  MoveL 3156 to (42.98, 34.27, 135) mm, rotated rx 180 ry 0 rz 180 deg; joints [33.282, 51.26, 5.095, -141.744, 62.408, -200.063]
  Call Extruder(29635.551)
  MoveL 3157 to (34.27, 42.98, 135) mm, rotated rx 180 ry 0 rz 180 deg; joints [34.874, 50.898, 5.796, -140.175, 63.224, -200.59]
  Call Extruder(29646.481)
  MoveL 3158 to (23.85, 49.52, 135) mm, rotated rx -180 ry 0 rz -180 deg; joints [36.387, 50.182, 7.18, -138.811, 64.267, -200.804]
  Call Extruder(29657.411)
  MoveL 3159 to (12.23, 53.59, 135) mm, rotated rx 180 ry 0 rz -180 deg; joints [37.766, 49.152, 9.175, -137.688, 65.475, -200.699]
  Call Extruder(29668.342)
  MoveL 3160 to (0, 54.97, 135) mm, rotated rx 180 ry 0 rz -180 deg; joints [38.954, 47.859, 11.678, -136.834, 66.781, -200.294]
  Call Extruder(29679.272)
  MoveL 3161 to (-12.23, 53.59, 135) mm, rotated rx 180 ry 0 rz -180 deg; joints [39.895, 46.371, 14.565, -136.276, 68.117, -199.62]
  Call Extruder(29690.202)
  MoveL 3162 to (-23.85, 49.53, 135) mm, rotated rx 180 ry 0 rz 180 deg; joints [40.528, 44.756, 17.699, -136.043, 69.421, -198.723]
  Call Extruder(29701.132)
  MoveL 3163 to (-34.27, 42.98, 135) mm, rotated rx 180 ry 0 rz 180 deg; joints [40.799, 43.092, 20.933, -136.165, 70.637, -197.658]
  Call Extruder(29712.062)
  MoveL 3164 to (-42.98, 34.27, 135) mm, rotated rx -180 ry 0 rz -180 deg; joints [40.659, 41.457, 24.115, -136.671, 71.717, -196.485]
  Call Extruder(29722.993)
  MoveL 3165 to (-49.53, 23.85, 135) mm, rotated rx 180 ry 0 rz 180 deg; joints [40.072, 39.93, 27.092, -137.58, 72.618, -195.268]
  Call Extruder(29733.923)
  MoveL 3166 to (-53.59, 12.23, 135) mm, rotated rx 180 ry 0 rz -180 deg; joints [39.031, 38.588, 29.712, -138.895, 73.308, -194.069]
  Call Extruder(29744.853)
  MoveL 3167 to (-54.97, 0, 135) mm, rotated rx 180 ry 0 rz -180 deg; joints [37.56, 37.502, 31.833, -140.584, 73.755, -192.948]
  Call Extruder(29750.379)
  MoveL 3168 to (-54.27, -6.18, 135) mm, rotated rx 180 ry 0 rz -180 deg; joints [36.644, 37.108, 32.604, -141.583, 73.846, -192.442]
  Set speed (130.0 mm/s)
  MoveL 3169 to (-49.9, -9.51, 135) mm, rotated rx -180 ry 0 rz 180 deg; joints [35.741, 37.302, 32.224, -142.469, 73.507, -192.303]
  MoveL 3170 to (2.97, -12.99, 135) mm, rotated rx 180 ry 0 rz -180 deg; joints [30.614, 42.764, 21.571, -146.715, 68.115, -193.75]
  Call Extruder(29755.042)
  Set speed (80.0 mm/s)
  MoveL 3171 to (5.78, -12.01, 135) mm, rotated rx -180 ry 0 rz -180 deg; joints [30.526, 43.158, 20.805, -146.725, 67.783, -193.936]
  Call Extruder(29759.706)
  MoveL 3172 to (8.31, -10.42, 135) mm, rotated rx -180 ry 0 rz -180 deg; joints [30.538, 43.562, 20.019, -146.625, 67.467, -194.168]
  Call Extruder(29764.370)
  MoveL 3173 to (10.42, -8.31, 135) mm, rotated rx 180 ry 0 rz 180 deg; joints [30.649, 43.956, 19.253, -146.423, 67.184, -194.435]
  Call Extruder(29769.034)
  MoveL 3174 to (12.01, -5.78, 135) mm, rotated rx 180 ry 0 rz -180 deg; joints [30.85, 44.321, 18.544, -146.131, 66.949, -194.725]
  Call Extruder(29773.697)
  MoveL 3175 to (12.99, -2.97, 135) mm, rotated rx 180 ry 0 rz -180 deg; joints [31.131, 44.637, 17.929, -145.765, 66.773, -195.022]
  Call Extruder(29778.361)
  MoveL 3176 to (13.33, 0, 135) mm, rotated rx 180 ry 0 rz -180 deg; joints [31.476, 44.891, 17.438, -145.344, 66.667, -195.312]
  Call Extruder(29783.025)
  MoveL 3177 to (12.99, 2.97, 135) mm, rotated rx 180 ry 0 rz -180 deg; joints [31.869, 45.068, 17.094, -144.89, 66.635, -195.58]
  Call Extruder(29787.689)
  MoveL 3178 to (12.01, 5.78, 135) mm, rotated rx 180 ry 0 rz -180 deg; joints [32.292, 45.16, 16.915, -144.425, 66.679, -195.81]
  Call Extruder(29792.352)
  MoveL 3179 to (10.42, 8.31, 135) mm, rotated rx 180 ry 0 rz 180 deg; joints [32.725, 45.162, 16.91, -143.971, 66.795, -195.991]
  Call Extruder(29797.017)
  MoveL 3180 to (8.31, 10.42, 135) mm, rotated rx -180 ry 0 rz -180 deg; joints [33.149, 45.075, 17.079, -143.549, 66.978, -196.112]
  Call Extruder(29801.680)
  MoveL 3181 to (5.78, 12.01, 135) mm, rotated rx 180 ry 0 rz -180 deg; joints [33.544, 44.903, 17.413, -143.177, 67.219, -196.167]
  Call Extruder(29806.344)
  MoveL 3182 to (2.97, 13, 135) mm, rotated rx 180 ry 0 rz -180 deg; joints [33.893, 44.654, 17.897, -142.874, 67.503, -196.154]
  Call Extruder(29811.008)
  MoveL 3183 to (0, 13.33, 135) mm, rotated rx 180 ry 0 rz 180 deg; joints [34.177, 44.341, 18.505, -142.652, 67.817, -196.073]
  Call Extruder(29815.672)
  MoveL 3184 to (-2.97, 12.99, 135) mm, rotated rx -180 ry 0 rz 180 deg; joints [34.384, 43.979, 19.209, -142.522, 68.145, -195.93]
  Call Extruder(29820.335)
  MoveL 3185 to (-5.78, 12.01, 135) mm, rotated rx 180 ry 0 rz 180 deg; joints [34.5, 43.586, 19.973, -142.491, 68.471, -195.731]
  Call Extruder(29824.999)
  MoveL 3186 to (-8.31, 10.42, 135) mm, rotated rx 180 ry 0 rz 180 deg; joints [34.518, 43.182, 20.759, -142.563, 68.779, -195.489]
  Call Extruder(29829.663)
  MoveL 3187 to (-10.42, 8.31, 135) mm, rotated rx 180 ry 0 rz -180 deg; joints [34.436, 42.787, 21.527, -142.735, 69.054, -195.215]
  Call Extruder(29834.327)
  MoveL 3188 to (-12.01, 5.78, 135) mm, rotated rx 180 ry 0 rz 180 deg; joints [34.254, 42.42, 22.24, -143.003, 69.283, -194.925]
  Call Extruder(29838.990)
  MoveL 3189 to (-12.99, 2.97, 135) mm, rotated rx 180 ry 0 rz 180 deg; joints [33.981, 42.101, 22.861, -143.353, 69.455, -194.632]
  Call Extruder(29843.654)
  MoveL 3190 to (-13.33, 0, 135) mm, rotated rx 180 ry 0 rz 180 deg; joints [33.63, 41.846, 23.359, -143.77, 69.562, -194.351]
  Call Extruder(29848.318)
  MoveL 3191 to (-13, -2.97, 135) mm, rotated rx 180 ry 0 rz -180 deg; joints [33.218, 41.667, 23.707, -144.233, 69.598, -194.096]
  Call Extruder(29852.982)
  MoveL 3192 to (-12.01, -5.78, 135) mm, rotated rx 180 ry 0 rz 180 deg; joints [32.767, 41.573, 23.889, -144.719, 69.561, -193.879]
  Call Extruder(29857.645)
  MoveL 3193 to (-10.42, -8.31, 135) mm, rotated rx 180 ry 0 rz 180 deg; joints [32.302, 41.571, 23.894, -145.201, 69.452, -193.708]
  Call Extruder(29862.310)
  MoveL 3194 to (-8.31, -10.42, 135) mm, rotated rx -180 ry 0 rz -180 deg; joints [31.85, 41.659, 23.723, -145.653, 69.277, -193.594]
  Call Extruder(29866.973)
  MoveL 3195 to (-5.78, -12.01, 135) mm, rotated rx 180 ry 0 rz 180 deg; joints [31.435, 41.833, 23.384, -146.05, 69.043, -193.539]
  Call Extruder(29871.637)
  MoveL 3196 to (-2.97, -12.99, 135) mm, rotated rx -180 ry 0 rz -180 deg; joints [31.079, 42.084, 22.894, -146.369, 68.762, -193.548]
  Call Extruder(29876.301)
  MoveL 3197 to (0, -13.33, 135) mm, rotated rx 180 ry 0 rz -180 deg; joints [30.801, 42.4, 22.279, -146.595, 68.447, -193.619]
  Call Extruder(29880.965)
  MoveL 3198 to (2.97, -12.99, 135) mm, rotated rx 180 ry 0 rz -180 deg; joints [30.614, 42.764, 21.571, -146.715, 68.115, -193.75]
  Set speed (130.0 mm/s)
  MoveL 3199 to (2.97, -12.99, 140) mm, rotated rx -180 ry 0 rz -180 deg; joints [30.614, 41.931, 21.714, -146.56, 67.539, -194.16]
  MoveL 3200 to (-26.25, -4.54, 140) mm, rotated rx 180 ry 0 rz 180 deg; joints [34.172, 39.236, 26.879, -143.407, 70.428, -193.968]
  Call Extruder(29883.197)
  Set speed (60.0 mm/s)
  MoveL 3201 to (-26.09, -5.96, 140) mm, rotated rx 180 ry 0 rz -180 deg; joints [33.969, 39.149, 27.045, -143.633, 70.443, -193.847]
  Call Extruder(29892.562)
  MoveL 3202 to (-24.12, -11.61, 140) mm, rotated rx 180 ry 0 rz -180 deg; joints [33.033, 38.956, 27.415, -144.635, 70.366, -193.413]
  Call Extruder(29901.927)
  MoveL 3203 to (-20.93, -16.69, 140) mm, rotated rx 180 ry 0 rz 180 deg; joints [32.066, 38.951, 27.426, -145.637, 70.148, -193.072]
  Call Extruder(29911.292)
  MoveL 3204 to (-16.69, -20.93, 140) mm, rotated rx 180 ry 0 rz 180 deg; joints [31.126, 39.133, 27.077, -146.578, 69.799, -192.838]
  Call Extruder(29920.657)
  MoveL 3205 to (-11.61, -24.11, 140) mm, rotated rx -180 ry 0 rz -180 deg; joints [30.272, 39.492, 26.388, -147.4, 69.334, -192.719]
  Call Extruder(29930.022)
  MoveL 3206 to (-5.96, -26.09, 140) mm, rotated rx 180 ry 0 rz 180 deg; joints [29.552, 40.01, 25.395, -148.055, 68.774, -192.721]
  Call Extruder(29939.387)
  MoveL 3207 to (0, -26.77, 140) mm, rotated rx 180 ry 0 rz 180 deg; joints [29.003, 40.659, 24.152, -148.507, 68.146, -192.846]
  Call Extruder(29948.752)
  MoveL 3208 to (5.96, -26.09, 140) mm, rotated rx 180 ry 0 rz 180 deg; joints [28.65, 41.404, 22.723, -148.733, 67.484, -193.09]
  Call Extruder(29958.117)
  MoveL 3209 to (11.61, -24.11, 140) mm, rotated rx 180 ry 0 rz 180 deg; joints [28.503, 42.209, 21.181, -148.728, 66.819, -193.446]
  Call Extruder(29967.482)
  MoveL 3210 to (16.69, -20.93, 140) mm, rotated rx -180 ry 0 rz -180 deg; joints [28.559, 43.032, 19.602, -148.497, 66.188, -193.898]
  Call Extruder(29976.847)
  MoveL 3211 to (20.93, -16.69, 140) mm, rotated rx 180 ry 0 rz 180 deg; joints [28.808, 43.834, 18.066, -148.06, 65.624, -194.429]
  Call Extruder(29986.212)
  MoveL 3212 to (24.12, -11.61, 140) mm, rotated rx 180 ry 0 rz -180 deg; joints [29.229, 44.574, 16.648, -147.446, 65.157, -195.014]
  Call Extruder(29995.577)
  MoveL 3213 to (26.09, -5.96, 140) mm, rotated rx 180 ry 0 rz -180 deg; joints [29.796, 45.217, 15.416, -146.693, 64.813, -195.622]
  Call Extruder(30004.942)
  MoveL 3214 to (26.77, 0, 140) mm, rotated rx 180 ry 0 rz -180 deg; joints [30.482, 45.73, 14.431, -145.841, 64.609, -196.223]
  Call Extruder(30014.307)
  MoveL 3215 to (26.09, 5.96, 140) mm, rotated rx 180 ry 0 rz -180 deg; joints [31.252, 46.09, 13.743, -144.933, 64.557, -196.781]
  Call Extruder(30023.672)
  MoveL 3216 to (24.12, 11.61, 140) mm, rotated rx 180 ry 0 rz -180 deg; joints [32.076, 46.277, 13.385, -144.015, 64.659, -197.265]
  Call Extruder(30033.037)
  MoveL 3217 to (20.93, 16.69, 140) mm, rotated rx 180 ry 0 rz -180 deg; joints [32.917, 46.282, 13.374, -143.126, 64.907, -197.646]
  Call Extruder(30042.402)
  MoveL 3218 to (16.69, 20.93, 140) mm, rotated rx 180 ry 0 rz 180 deg; joints [33.742, 46.106, 13.712, -142.305, 65.288, -197.903]
  Call Extruder(30051.767)
  MoveL 3219 to (11.61, 24.12, 140) mm, rotated rx 180 ry 0 rz 180 deg; joints [34.517, 45.756, 14.382, -141.585, 65.779, -198.022]
  Call Extruder(30061.132)
  MoveL 3220 to (5.96, 26.09, 140) mm, rotated rx 180 ry 0 rz 180 deg; joints [35.208, 45.251, 15.351, -140.995, 66.354, -197.997]
  Call Extruder(30070.497)
  MoveL 3221 to (0, 26.77, 140) mm, rotated rx 180 ry 0 rz 180 deg; joints [35.784, 44.615, 16.569, -140.557, 66.983, -197.831]
  Call Extruder(30079.862)
  MoveL 3222 to (-5.96, 26.09, 140) mm, rotated rx 180 ry 0 rz 180 deg; joints [36.214, 43.879, 17.979, -140.292, 67.633, -197.537]
  Call Extruder(30089.227)
  MoveL 3223 to (-11.61, 24.12, 140) mm, rotated rx 180 ry 0 rz -180 deg; joints [36.473, 43.08, 19.51, -140.215, 68.273, -197.132]
  Call Extruder(30098.591)
  MoveL 3224 to (-16.69, 20.93, 140) mm, rotated rx 180 ry 0 rz 180 deg; joints [36.542, 42.257, 21.088, -140.334, 68.874, -196.64]
  Call Extruder(30107.957)
  MoveL 3225 to (-20.93, 16.69, 140) mm, rotated rx 180 ry 0 rz -180 deg; joints [36.407, 41.451, 22.634, -140.652, 69.406, -196.087]
  Call Extruder(30117.322)
  MoveL 3226 to (-24.12, 11.61, 140) mm, rotated rx 180 ry 0 rz 180 deg; joints [36.065, 40.7, 24.072, -141.163, 69.847, -195.502]
  Call Extruder(30126.686)
  MoveL 3227 to (-26.09, 5.96, 140) mm, rotated rx 180 ry 0 rz 180 deg; joints [35.528, 40.045, 25.328, -141.851, 70.176, -194.916]
  Call Extruder(30136.051)
  MoveL 3228 to (-26.77, 0, 140) mm, rotated rx 180 ry 0 rz 180 deg; joints [34.817, 39.519, 26.337, -142.688, 70.378, -194.355]
  Call Extruder(30140.840)
  MoveL 3229 to (-26.42, -3.05, 140) mm, rotated rx 180 ry 0 rz -180 deg; joints [34.385, 39.328, 26.702, -143.17, 70.412, -194.095]
  Set speed (130.0 mm/s)
  MoveL 3230 to (-41.86, -6.29, 140) mm, rotated rx 180 ry 0 rz -180 deg; joints [35.393, 37.441, 30.319, -142.491, 72.029, -193.324]
  Call Extruder(30145.838)
  Set speed (60.0 mm/s)
  MoveL 3231 to (-41.5, -9.47, 140) mm, rotated rx 180 ry 0 rz -180 deg; joints [34.924, 37.244, 30.696, -143.006, 72.065, -193.061]
  Call Extruder(30160.734)
  MoveL 3232 to (-38.36, -18.47, 140) mm, rotated rx 180 ry 0 rz -180 deg; joints [33.373, 36.932, 31.296, -144.652, 71.955, -192.392]
  Call Extruder(30175.630)
  MoveL 3233 to (-33.29, -26.54, 140) mm, rotated rx 180 ry 0 rz 180 deg; joints [31.763, 36.923, 31.313, -146.31, 71.624, -191.869]
  Call Extruder(30190.525)
  MoveL 3234 to (-26.54, -33.29, 140) mm, rotated rx -180 ry 0 rz 180 deg; joints [30.206, 37.218, 30.748, -147.87, 71.081, -191.509]
  Call Extruder(30205.421)
  MoveL 3235 to (-18.47, -38.36, 140) mm, rotated rx 180 ry 0 rz 180 deg; joints [28.808, 37.799, 29.633, -149.225, 70.349, -191.325]
  Call Extruder(30220.317)
  MoveL 3236 to (-9.47, -41.5, 140) mm, rotated rx 180 ry 0 rz 180 deg; joints [27.654, 38.634, 28.033, -150.288, 69.462, -191.321]
  Call Extruder(30235.213)
  MoveL 3237 to (0, -42.57, 140) mm, rotated rx -180 ry 0 rz -180 deg; joints [26.805, 39.675, 26.038, -151, 68.462, -191.502]
  Call Extruder(30250.109)
  MoveL 3238 to (9.47, -41.5, 140) mm, rotated rx 180 ry 0 rz -180 deg; joints [26.29, 40.867, 23.753, -151.331, 67.401, -191.866]
  Call Extruder(30265.004)
  MoveL 3239 to (18.47, -38.36, 140) mm, rotated rx 180 ry 0 rz 180 deg; joints [26.114, 42.149, 21.296, -151.277, 66.333, -192.407]
  Call Extruder(30279.900)
  MoveL 3240 to (26.54, -33.29, 140) mm, rotated rx -180 ry 0 rz 180 deg; joints [26.262, 43.457, 18.787, -150.858, 65.315, -193.108]
  Call Extruder(30294.796)
  MoveL 3241 to (33.28, -26.54, 140) mm, rotated rx 180 ry 0 rz 180 deg; joints [26.703, 44.73, 16.349, -150.114, 64.404, -193.944]
  Call Extruder(30309.692)
  MoveL 3242 to (38.36, -18.47, 140) mm, rotated rx 180 ry 0 rz 180 deg; joints [27.4, 45.905, 14.097, -149.098, 63.648, -194.878]
  Call Extruder(30324.587)
  MoveL 3243 to (41.51, -9.47, 140) mm, rotated rx 180 ry 0 rz 180 deg; joints [28.309, 46.926, 12.141, -147.873, 63.091, -195.865]
  Call Extruder(30339.483)
  MoveL 3244 to (42.57, 0, 140) mm, rotated rx 180 ry 0 rz 180 deg; joints [29.382, 47.743, 10.575, -146.508, 62.765, -196.847]
  Call Extruder(30354.379)
  MoveL 3245 to (41.5, 9.47, 140) mm, rotated rx 180 ry 0 rz -180 deg; joints [30.575, 48.315, 9.478, -145.076, 62.686, -197.765]
  Call Extruder(30369.275)
  MoveL 3246 to (38.36, 18.47, 140) mm, rotated rx -180 ry 0 rz -180 deg; joints [31.839, 48.614, 8.907, -143.643, 62.858, -198.563]
  Call Extruder(30384.171)
  MoveL 3247 to (33.29, 26.54, 140) mm, rotated rx 180 ry 0 rz -180 deg; joints [33.128, 48.622, 8.89, -142.273, 63.269, -199.188]
  Call Extruder(30399.067)
  MoveL 3248 to (26.54, 33.28, 140) mm, rotated rx -180 ry 0 rz -180 deg; joints [34.394, 48.341, 9.43, -141.018, 63.891, -199.603]
  Call Extruder(30413.962)
  MoveL 3249 to (18.47, 38.36, 140) mm, rotated rx -180 ry 0 rz 180 deg; joints [35.592, 47.784, 10.496, -139.922, 64.689, -199.785]
  Call Extruder(30428.858)
  MoveL 3250 to (9.47, 41.51, 140) mm, rotated rx 180 ry 0 rz -180 deg; joints [36.675, 46.98, 12.037, -139.022, 65.614, -199.73]
  Call Extruder(30443.754)
  MoveL 3251 to (0, 42.57, 140) mm, rotated rx 180 ry 0 rz 180 deg; joints [37.594, 45.97, 13.973, -138.345, 66.618, -199.445]
  Call Extruder(30458.650)
  MoveL 3252 to (-9.47, 41.51, 140) mm, rotated rx -180 ry 0 rz -180 deg; joints [38.304, 44.802, 16.21, -137.918, 67.648, -198.953]
  Call Extruder(30473.545)
  MoveL 3253 to (-18.47, 38.36, 140) mm, rotated rx 180 ry 0 rz 180 deg; joints [38.762, 43.534, 18.641, -137.763, 68.656, -198.286]
  Call Extruder(30488.441)
  MoveL 3254 to (-26.54, 33.29, 140) mm, rotated rx 180 ry 0 rz -180 deg; joints [38.928, 42.226, 21.148, -137.901, 69.596, -197.485]
  Call Extruder(30503.337)
  MoveL 3255 to (-33.28, 26.54, 140) mm, rotated rx 180 ry 0 rz 180 deg; joints [38.772, 40.941, 23.612, -138.346, 70.427, -196.594]
  Call Extruder(30518.233)
  MoveL 3256 to (-38.36, 18.47, 140) mm, rotated rx 180 ry 0 rz 180 deg; joints [38.277, 39.742, 25.91, -139.103, 71.116, -195.66]
  Call Extruder(30533.129)
  MoveL 3257 to (-41.51, 9.47, 140) mm, rotated rx 180 ry 0 rz -180 deg; joints [37.447, 38.69, 27.925, -140.159, 71.633, -194.731]
  Call Extruder(30548.024)
  MoveL 3258 to (-42.57, 0, 140) mm, rotated rx 180 ry 0 rz -180 deg; joints [36.31, 37.842, 29.551, -141.48, 71.955, -193.851]
  Call Extruder(30555.579)
  MoveL 3259 to (-42.03, -4.8, 140) mm, rotated rx -180 ry 0 rz 180 deg; joints [35.612, 37.535, 30.139, -142.25, 72.011, -193.448]
  Set speed (130.0 mm/s)
  MoveL 3260 to (-54.1, -7.67, 140) mm, rotated rx 180 ry 0 rz -180 deg; joints [36.421, 36.076, 32.935, -141.682, 73.249, -192.831]
  Call Extruder(30559.651)
  Set speed (30.0 mm/s)
  MoveL 3261 to (-53.59, -12.23, 140) mm, rotated rx 180 ry 0 rz -180 deg; joints [35.732, 35.79, 33.484, -142.433, 73.304, -192.461]
  Call Extruder(30570.582)
  MoveL 3262 to (-49.53, -23.85, 140) mm, rotated rx 180 ry 0 rz -180 deg; joints [33.663, 35.379, 34.271, -144.613, 73.176, -191.618]
  Call Extruder(30581.512)
  MoveL 3263 to (-42.98, -34.27, 140) mm, rotated rx 180 ry 0 rz 180 deg; joints [31.506, 35.367, 34.294, -146.828, 72.762, -190.963]
  Call Extruder(30592.442)
  MoveL 3264 to (-34.27, -42.98, 140) mm, rotated rx -180 ry 0 rz 180 deg; joints [29.427, 35.755, 33.55, -148.91, 72.074, -190.514]
  Call Extruder(30603.372)
  MoveL 3265 to (-23.85, -49.53, 140) mm, rotated rx -180 ry 0 rz 180 deg; joints [27.581, 36.518, 32.089, -150.707, 71.136, -190.281]
  Call Extruder(30614.302)
  MoveL 3266 to (-12.23, -53.59, 140) mm, rotated rx -180 ry 0 rz -180 deg; joints [26.087, 37.608, 29.999, -152.097, 69.992, -190.269]
  Call Extruder(30625.233)
  MoveL 3267 to (0, -54.97, 140) mm, rotated rx 180 ry 0 rz 180 deg; joints [25.019, 38.963, 27.403, -153.004, 68.698, -190.485]
  Call Extruder(30634.985)
  MoveL 3268 to (10.91, -53.74, 140) mm, rotated rx 180 ry 0 rz 180 deg; joints [24.47, 40.34, 24.764, -153.357, 67.47, -190.882]
  Call Extruder(30636.163)
  MoveL 3269 to (12.23, -53.59, 140) mm, rotated rx -180 ry 0 rz -180 deg; joints [24.406, 40.508, 24.441, -153.396, 67.32, -190.931]
  Call Extruder(30647.093)
  MoveL 3270 to (23.85, -49.52, 140) mm, rotated rx -180 ry 0 rz -180 deg; joints [24.239, 42.165, 21.265, -153.279, 65.93, -191.603]
  Call Extruder(30658.023)
  MoveL 3271 to (34.27, -42.98, 140) mm, rotated rx -180 ry 0 rz -180 deg; joints [24.487, 43.853, 18.029, -152.688, 64.603, -192.488]
  Call Extruder(30668.953)
  MoveL 3272 to (42.98, -34.27, 140) mm, rotated rx -180 ry 0 rz -180 deg; joints [25.101, 45.494, 14.885, -151.68, 63.411, -193.561]
  Call Extruder(30679.884)
  MoveL 3273 to (49.52, -23.85, 140) mm, rotated rx 180 ry 0 rz -180 deg; joints [26.025, 47.01, 11.979, -150.33, 62.422, -194.775]
  Call Extruder(30690.814)
  MoveL 3274 to (53.59, -12.23, 140) mm, rotated rx 180 ry 0 rz -180 deg; joints [27.2, 48.33, 9.451, -148.722, 61.692, -196.07]
  Call Extruder(30701.744)
  MoveL 3275 to (54.97, 0, 140) mm, rotated rx 180 ry 0 rz 180 deg; joints [28.57, 49.388, 7.423, -146.949, 61.266, -197.37]
  Call Extruder(30712.674)
  MoveL 3276 to (53.59, 12.23, 140) mm, rotated rx -180 ry 0 rz -180 deg; joints [30.077, 50.131, 6.001, -145.105, 61.167, -198.591]
  Call Extruder(30723.604)
  MoveL 3277 to (49.53, 23.85, 140) mm, rotated rx 180 ry 0 rz -180 deg; joints [31.665, 50.518, 5.259, -143.28, 61.4, -199.65]
  Call Extruder(30734.535)
  MoveL 3278 to (42.98, 34.27, 140) mm, rotated rx 180 ry 0 rz -180 deg; joints [33.282, 50.53, 5.237, -141.551, 61.947, -200.476]
  Call Extruder(30745.465)
  MoveL 3279 to (34.27, 42.98, 140) mm, rotated rx 180 ry 0 rz -180 deg; joints [34.874, 50.164, 5.938, -139.981, 62.77, -201.017]
  Call Extruder(30756.395)
  MoveL 3280 to (23.85, 49.53, 140) mm, rotated rx 180 ry 0 rz 180 deg; joints [36.387, 49.441, 7.322, -138.619, 63.817, -201.244]
  Call Extruder(30767.325)
  MoveL 3281 to (12.23, 53.59, 140) mm, rotated rx 180 ry 0 rz -180 deg; joints [37.766, 48.4, 9.316, -137.498, 65.025, -201.153]
  Call Extruder(30778.255)
  MoveL 3282 to (0, 54.97, 140) mm, rotated rx 180 ry 0 rz 180 deg; joints [38.954, 47.094, 11.819, -136.648, 66.326, -200.76]
  Call Extruder(30789.186)
  MoveL 3283 to (-12.23, 53.59, 140) mm, rotated rx 180 ry 0 rz 180 deg; joints [39.895, 45.587, 14.706, -136.096, 67.653, -200.1]
  Call Extruder(30800.116)
  MoveL 3284 to (-23.85, 49.52, 140) mm, rotated rx 180 ry 0 rz -180 deg; joints [40.528, 43.952, 17.84, -135.868, 68.944, -199.216]
  Call Extruder(30811.046)
  MoveL 3285 to (-34.27, 42.98, 140) mm, rotated rx 180 ry 0 rz -180 deg; joints [40.799, 42.264, 21.075, -135.995, 70.143, -198.163]
  Call Extruder(30821.976)
  MoveL 3286 to (-42.98, 34.27, 140) mm, rotated rx 180 ry 0 rz 180 deg; joints [40.659, 40.603, 24.259, -136.507, 71.2, -197]
  Call Extruder(30832.906)
  MoveL 3287 to (-49.53, 23.85, 140) mm, rotated rx 180 ry 0 rz -180 deg; joints [40.072, 39.049, 27.237, -137.422, 72.076, -195.789]
  Call Extruder(30843.837)
  MoveL 3288 to (-53.59, 12.23, 140) mm, rotated rx 180 ry 0 rz -180 deg; joints [39.031, 37.681, 29.859, -138.742, 72.736, -194.592]
  Call Extruder(30854.767)
  MoveL 3289 to (-54.97, 0, 140) mm, rotated rx 180 ry 0 rz -180 deg; joints [37.56, 36.574, 31.982, -140.437, 73.153, -193.466]
  Call Extruder(30860.292)
  MoveL 3290 to (-54.27, -6.18, 140) mm, rotated rx 180 ry 0 rz 180 deg; joints [36.644, 36.171, 32.753, -141.438, 73.23, -192.953]
  Set speed (130.0 mm/s)
  MoveL 3291 to (-49.9, -9.51, 140) mm, rotated rx -180 ry 0 rz -180 deg; joints [35.741, 36.369, 32.374, -142.324, 72.886, -192.802]
  MoveL 3292 to (2.97, -12.99, 140) mm, rotated rx -180 ry 0 rz -180 deg; joints [30.614, 41.931, 21.714, -146.56, 67.539, -194.16]
  Call Extruder(30864.956)
  Set speed (80.0 mm/s)
  MoveL 3293 to (5.78, -12.01, 140) mm, rotated rx 180 ry 0 rz 180 deg; joints [30.526, 42.331, 20.947, -146.569, 67.211, -194.344]
  Call Extruder(30869.620)
  MoveL 3294 to (8.31, -10.42, 140) mm, rotated rx 180 ry 0 rz -180 deg; joints [30.538, 42.741, 20.16, -146.468, 66.9, -194.574]
  Call Extruder(30874.284)
  MoveL 3295 to (10.42, -8.31, 140) mm, rotated rx 180 ry 0 rz 180 deg; joints [30.649, 43.141, 19.394, -146.264, 66.623, -194.841]
  Call Extruder(30878.947)
  MoveL 3296 to (12.01, -5.78, 140) mm, rotated rx -180 ry 0 rz 180 deg; joints [30.85, 43.51, 18.686, -145.97, 66.394, -195.131]
  Call Extruder(30883.611)
  MoveL 3297 to (12.99, -2.97, 140) mm, rotated rx 180 ry 0 rz 180 deg; joints [31.131, 43.831, 18.071, -145.602, 66.225, -195.431]
  Call Extruder(30888.275)
  MoveL 3298 to (13.33, 0, 140) mm, rotated rx -180 ry 0 rz 180 deg; joints [31.476, 44.088, 17.579, -145.18, 66.124, -195.724]
  Call Extruder(30892.939)
  MoveL 3299 to (13, 2.97, 140) mm, rotated rx 180 ry 0 rz -180 deg; joints [31.869, 44.267, 17.235, -144.724, 66.096, -195.994]
  Call Extruder(30897.602)
  MoveL 3300 to (12.01, 5.78, 140) mm, rotated rx 180 ry 0 rz 180 deg; joints [32.292, 44.361, 17.056, -144.258, 66.144, -196.228]
  Call Extruder(30902.266)
  MoveL 3301 to (10.42, 8.31, 140) mm, rotated rx 180 ry 0 rz 180 deg; joints [32.725, 44.363, 17.051, -143.803, 66.264, -196.413]
  Call Extruder(30906.930)
  MoveL 3302 to (8.31, 10.42, 140) mm, rotated rx 180 ry 0 rz 180 deg; joints [33.149, 44.275, 17.22, -143.38, 66.449, -196.539]
  Call Extruder(30911.594)
  MoveL 3303 to (5.78, 12.01, 140) mm, rotated rx 180 ry 0 rz -180 deg; joints [33.544, 44.101, 17.555, -143.009, 66.69, -196.599]
  Call Extruder(30916.257)
  MoveL 3304 to (2.97, 13, 140) mm, rotated rx 180 ry 0 rz -180 deg; joints [33.893, 43.848, 18.038, -142.705, 66.974, -196.59]
  Call Extruder(30920.921)
  MoveL 3305 to (0, 13.33, 140) mm, rotated rx 180 ry 0 rz 180 deg; joints [34.177, 43.531, 18.647, -142.484, 67.286, -196.513]
  Call Extruder(30925.585)
  MoveL 3306 to (-2.97, 13, 140) mm, rotated rx 180 ry 0 rz 180 deg; joints [34.384, 43.164, 19.351, -142.355, 67.611, -196.373]
  Call Extruder(30930.249)
  MoveL 3307 to (-5.78, 12.01, 140) mm, rotated rx -180 ry 0 rz 180 deg; joints [34.5, 42.765, 20.115, -142.326, 67.933, -196.177]
  Call Extruder(30934.913)
  MoveL 3308 to (-8.31, 10.42, 140) mm, rotated rx 180 ry 0 rz 180 deg; joints [34.518, 42.355, 20.901, -142.399, 68.236, -195.937]
  Call Extruder(30939.577)
  MoveL 3309 to (-10.42, 8.31, 140) mm, rotated rx 180 ry 0 rz 180 deg; joints [34.436, 41.954, 21.67, -142.573, 68.505, -195.665]
  Call Extruder(30944.240)
  MoveL 3310 to (-12.01, 5.78, 140) mm, rotated rx 180 ry 0 rz -180 deg; joints [34.254, 41.582, 22.383, -142.842, 68.728, -195.374]
  Call Extruder(30948.904)
  MoveL 3311 to (-13, 2.97, 140) mm, rotated rx -180 ry 0 rz 180 deg; joints [33.981, 41.258, 23.004, -143.193, 68.894, -195.08]
  Call Extruder(30953.568)
  MoveL 3312 to (-13.33, 0, 140) mm, rotated rx 180 ry 0 rz 180 deg; joints [33.63, 40.998, 23.502, -143.612, 68.994, -194.797]
  Call Extruder(30958.232)
  MoveL 3313 to (-13, -2.97, 140) mm, rotated rx -180 ry 0 rz -180 deg; joints [33.218, 40.816, 23.851, -144.077, 69.025, -194.539]
  Call Extruder(30962.895)
  MoveL 3314 to (-12.01, -5.78, 140) mm, rotated rx 180 ry 0 rz -180 deg; joints [32.767, 40.721, 24.033, -144.564, 68.983, -194.317]
  Call Extruder(30967.559)
  MoveL 3315 to (-10.42, -8.31, 140) mm, rotated rx -180 ry 0 rz -180 deg; joints [32.302, 40.718, 24.038, -145.047, 68.871, -194.142]
  Call Extruder(30972.223)
  MoveL 3316 to (-8.31, -10.42, 140) mm, rotated rx -180 ry 0 rz -180 deg; joints [31.85, 40.808, 23.866, -145.499, 68.694, -194.022]
  Call Extruder(30976.887)
  MoveL 3317 to (-5.78, -12.01, 140) mm, rotated rx 180 ry 0 rz -180 deg; joints [31.435, 40.985, 23.527, -145.896, 68.459, -193.962]
  Call Extruder(30981.550)
  MoveL 3318 to (-2.97, -12.99, 140) mm, rotated rx -180 ry 0 rz -180 deg; joints [31.079, 41.24, 23.037, -146.216, 68.179, -193.966]
  Call Extruder(30986.214)
  MoveL 3319 to (0, -13.33, 140) mm, rotated rx -180 ry 0 rz -180 deg; joints [30.801, 41.561, 22.422, -146.441, 67.867, -194.033]
  Call Extruder(30990.878)
  MoveL 3320 to (2.97, -12.99, 140) mm, rotated rx -180 ry 0 rz -180 deg; joints [30.614, 41.931, 21.714, -146.56, 67.539, -194.16]
  Set speed (130.0 mm/s)
  MoveL 3321 to (2.97, -12.99, 145) mm, rotated rx 180 ry 0 rz 180 deg; joints [30.614, 41.106, 21.839, -146.398, 66.955, -194.58]
  MoveL 3322 to (-26.25, -4.54, 145) mm, rotated rx 180 ry 0 rz 180 deg; joints [34.172, 38.367, 27.006, -143.247, 69.833, -194.439]
  Call Extruder(30993.111)
  Set speed (60.0 mm/s)
  MoveL 3323 to (-26.09, -5.96, 145) mm, rotated rx 180 ry 0 rz -180 deg; joints [33.969, 38.278, 27.173, -143.474, 69.845, -194.317]
  Call Extruder(31002.476)
  MoveL 3324 to (-24.12, -11.61, 145) mm, rotated rx 180 ry 0 rz -180 deg; joints [33.033, 38.082, 27.543, -144.478, 69.757, -193.874]
  Call Extruder(31011.841)
  MoveL 3325 to (-20.93, -16.69, 145) mm, rotated rx -180 ry 0 rz 180 deg; joints [32.066, 38.076, 27.554, -145.482, 69.532, -193.522]
  Call Extruder(31021.206)
  MoveL 3326 to (-16.69, -20.93, 145) mm, rotated rx 180 ry 0 rz 180 deg; joints [31.126, 38.262, 27.205, -146.424, 69.179, -193.276]
  Call Extruder(31030.571)
  MoveL 3327 to (-11.61, -24.11, 145) mm, rotated rx 180 ry 0 rz 180 deg; joints [30.272, 38.628, 26.515, -147.247, 68.713, -193.145]
  Call Extruder(31039.936)
  MoveL 3328 to (-5.96, -26.09, 145) mm, rotated rx -180 ry 0 rz -180 deg; joints [29.552, 39.154, 25.522, -147.902, 68.155, -193.137]
  Call Extruder(31049.301)
  MoveL 3329 to (0, -26.77, 145) mm, rotated rx 180 ry 0 rz -180 deg; joints [29.003, 39.814, 24.278, -148.353, 67.534, -193.253]
  Call Extruder(31058.666)
  MoveL 3330 to (5.96, -26.09, 145) mm, rotated rx -180 ry 0 rz -180 deg; joints [28.65, 40.571, 22.848, -148.578, 66.879, -193.49]
  Call Extruder(31068.031)
  MoveL 3331 to (11.61, -24.11, 145) mm, rotated rx 180 ry 0 rz 180 deg; joints [28.503, 41.388, 21.306, -148.57, 66.225, -193.84]
  Call Extruder(31077.396)
  MoveL 3332 to (16.69, -20.93, 145) mm, rotated rx 180 ry 0 rz -180 deg; joints [28.559, 42.223, 19.727, -148.336, 65.605, -194.291]
  Call Extruder(31086.761)
  MoveL 3333 to (20.93, -16.69, 145) mm, rotated rx 180 ry 0 rz 180 deg; joints [28.808, 43.036, 18.191, -147.896, 65.053, -194.822]
  Call Extruder(31096.126)
  MoveL 3334 to (24.12, -11.61, 145) mm, rotated rx 180 ry 0 rz -180 deg; joints [29.229, 43.786, 16.772, -147.278, 64.598, -195.409]
  Call Extruder(31105.490)
  MoveL 3335 to (26.09, -5.96, 145) mm, rotated rx 180 ry 0 rz -180 deg; joints [29.796, 44.437, 15.54, -146.521, 64.265, -196.022]
  Call Extruder(31114.856)
  MoveL 3336 to (26.77, 0, 145) mm, rotated rx 180 ry 0 rz -180 deg; joints [30.482, 44.957, 14.555, -145.665, 64.072, -196.629]
  Call Extruder(31124.221)
  MoveL 3337 to (26.09, 5.96, 145) mm, rotated rx 180 ry 0 rz 180 deg; joints [31.252, 45.32, 13.867, -144.754, 64.03, -197.194]
  Call Extruder(31133.585)
  MoveL 3338 to (24.11, 11.61, 145) mm, rotated rx -180 ry 0 rz -180 deg; joints [32.076, 45.51, 13.508, -143.833, 64.139, -197.685]
  Call Extruder(31142.950)
  MoveL 3339 to (20.93, 16.69, 145) mm, rotated rx -180 ry 0 rz -180 deg; joints [32.917, 45.515, 13.498, -142.943, 64.394, -198.074]
  Call Extruder(31152.316)
  MoveL 3340 to (16.69, 20.93, 145) mm, rotated rx 180 ry 0 rz 180 deg; joints [33.742, 45.337, 13.836, -142.121, 64.778, -198.339]
  Call Extruder(31161.681)
  MoveL 3341 to (11.61, 24.12, 145) mm, rotated rx 180 ry 0 rz 180 deg; joints [34.517, 44.983, 14.506, -141.401, 65.271, -198.466]
  Call Extruder(31171.045)
  MoveL 3342 to (5.96, 26.09, 145) mm, rotated rx 180 ry 0 rz -180 deg; joints [35.208, 44.471, 15.475, -140.811, 65.845, -198.449]
  Call Extruder(31180.410)
  MoveL 3343 to (0, 26.77, 145) mm, rotated rx -180 ry 0 rz 180 deg; joints [35.784, 43.827, 16.693, -140.375, 66.471, -198.291]
  Call Extruder(31189.776)
  MoveL 3344 to (-5.96, 26.09, 145) mm, rotated rx 180 ry 0 rz -180 deg; joints [36.214, 43.082, 18.103, -140.113, 67.116, -198.004]
  Call Extruder(31199.140)
  MoveL 3345 to (-11.61, 24.12, 145) mm, rotated rx 180 ry 0 rz 180 deg; joints [36.473, 42.272, 19.635, -140.038, 67.749, -197.605]
  Call Extruder(31208.505)
  MoveL 3346 to (-16.69, 20.93, 145) mm, rotated rx 180 ry 0 rz -180 deg; joints [36.542, 41.437, 21.213, -140.16, 68.339, -197.117]
  Call Extruder(31217.870)
  MoveL 3347 to (-20.93, 16.69, 145) mm, rotated rx 180 ry 0 rz 180 deg; joints [36.407, 40.618, 22.76, -140.481, 68.86, -196.568]
  Call Extruder(31227.235)
  MoveL 3348 to (-24.12, 11.61, 145) mm, rotated rx 180 ry 0 rz 180 deg; joints [36.065, 39.856, 24.198, -140.995, 69.288, -195.984]
  Call Extruder(31236.600)
  MoveL 3349 to (-26.09, 5.96, 145) mm, rotated rx 180 ry 0 rz 180 deg; joints [35.528, 39.19, 25.455, -141.686, 69.604, -195.396]
  Call Extruder(31245.965)
  MoveL 3350 to (-26.77, 0, 145) mm, rotated rx 180 ry 0 rz 180 deg; joints [34.817, 38.654, 26.465, -142.526, 69.793, -194.832]
  Call Extruder(31250.754)
  MoveL 3351 to (-26.42, -3.05, 145) mm, rotated rx 180 ry 0 rz 180 deg; joints [34.385, 38.461, 26.83, -143.009, 69.82, -194.567]
  Set speed (130.0 mm/s)
  MoveL 3352 to (-41.86, -6.29, 145) mm, rotated rx 180 ry 0 rz -180 deg; joints [35.393, 36.539, 30.448, -142.335, 71.416, -193.821]
  Call Extruder(31255.752)
  Set speed (60.0 mm/s)
  MoveL 3353 to (-41.5, -9.47, 145) mm, rotated rx 180 ry 0 rz -180 deg; joints [34.924, 36.338, 30.826, -142.852, 71.446, -193.554]
  Call Extruder(31270.647)
  MoveL 3354 to (-38.36, -18.47, 145) mm, rotated rx 180 ry 0 rz -180 deg; joints [33.373, 36.019, 31.426, -144.501, 71.317, -192.87]
  Call Extruder(31285.543)
  MoveL 3355 to (-33.29, -26.54, 145) mm, rotated rx 180 ry 0 rz 180 deg; joints [31.763, 36.009, 31.443, -146.163, 70.973, -192.328]
  Call Extruder(31300.439)
  MoveL 3356 to (-26.54, -33.29, 145) mm, rotated rx -180 ry 0 rz 180 deg; joints [30.206, 36.31, 30.877, -147.725, 70.423, -191.948]
  Call Extruder(31315.335)
  MoveL 3357 to (-18.47, -38.36, 145) mm, rotated rx -180 ry 0 rz -180 deg; joints [28.808, 36.903, 29.762, -149.082, 69.691, -191.743]
  Call Extruder(31330.231)
  MoveL 3358 to (-9.47, -41.5, 145) mm, rotated rx 180 ry 0 rz -180 deg; joints [27.654, 37.754, 28.161, -150.146, 68.809, -191.721]
  Call Extruder(31345.127)
  MoveL 3359 to (0, -42.57, 145) mm, rotated rx 180 ry 0 rz -180 deg; joints [26.805, 38.813, 26.165, -150.857, 67.82, -191.887]
  Call Extruder(31360.022)
  MoveL 3360 to (9.47, -41.5, 145) mm, rotated rx -180 ry 0 rz 180 deg; joints [26.29, 40.025, 23.879, -151.185, 66.773, -192.24]
  Call Extruder(31374.918)
  MoveL 3361 to (18.47, -38.36, 145) mm, rotated rx 180 ry 0 rz 180 deg; joints [26.114, 41.327, 21.421, -151.128, 65.722, -192.774]
  Call Extruder(31389.814)
  MoveL 3362 to (26.54, -33.28, 145) mm, rotated rx 180 ry 0 rz 180 deg; joints [26.262, 42.654, 18.912, -150.704, 64.723, -193.473]
  Call Extruder(31404.710)
  MoveL 3363 to (33.28, -26.54, 145) mm, rotated rx 180 ry 0 rz 180 deg; joints [26.703, 43.944, 16.473, -149.954, 63.83, -194.311]
  Call Extruder(31419.606)
  MoveL 3364 to (38.36, -18.47, 145) mm, rotated rx -180 ry 0 rz 180 deg; joints [27.4, 45.133, 14.221, -148.931, 63.093, -195.251]
  Call Extruder(31434.501)
  MoveL 3365 to (41.5, -9.47, 145) mm, rotated rx 180 ry 0 rz -180 deg; joints [28.309, 46.166, 12.264, -147.699, 62.554, -196.246]
  Call Extruder(31449.397)
  MoveL 3366 to (42.57, 0, 145) mm, rotated rx 180 ry 0 rz 180 deg; joints [29.382, 46.993, 10.699, -146.328, 62.243, -197.238]
  Call Extruder(31464.293)
  MoveL 3367 to (41.51, 9.47, 145) mm, rotated rx -180 ry 0 rz -180 deg; joints [30.575, 47.571, 9.602, -144.89, 62.178, -198.167]
  Call Extruder(31479.189)
  MoveL 3368 to (38.36, 18.47, 145) mm, rotated rx 180 ry 0 rz -180 deg; joints [31.839, 47.873, 9.031, -143.453, 62.362, -198.975]
  Call Extruder(31494.084)
  MoveL 3369 to (33.28, 26.54, 145) mm, rotated rx -180 ry 0 rz -180 deg; joints [33.128, 47.881, 9.014, -142.08, 62.781, -199.612]
  Call Extruder(31508.980)
  MoveL 3370 to (26.54, 33.29, 145) mm, rotated rx 180 ry 0 rz 180 deg; joints [34.394, 47.597, 9.554, -140.824, 63.41, -200.039]
  Call Extruder(31523.876)
  MoveL 3371 to (18.47, 38.36, 145) mm, rotated rx 180 ry 0 rz -180 deg; joints [35.592, 47.034, 10.62, -139.729, 64.21, -200.233]
  Call Extruder(31538.772)
  MoveL 3372 to (9.47, 41.51, 145) mm, rotated rx 180 ry 0 rz 180 deg; joints [36.675, 46.221, 12.161, -138.83, 65.135, -200.189]
  Call Extruder(31553.668)
  MoveL 3373 to (0, 42.57, 145) mm, rotated rx -180 ry 0 rz 180 deg; joints [37.594, 45.199, 14.097, -138.157, 66.135, -199.915]
  Call Extruder(31568.564)
  MoveL 3374 to (-9.47, 41.51, 145) mm, rotated rx 180 ry 0 rz -180 deg; joints [38.304, 44.017, 16.334, -137.733, 67.158, -199.434]
  Call Extruder(31583.459)
  MoveL 3375 to (-18.47, 38.36, 145) mm, rotated rx 180 ry 0 rz -180 deg; joints [38.762, 42.732, 18.765, -137.583, 68.155, -198.777]
  Call Extruder(31598.355)
  MoveL 3376 to (-26.54, 33.28, 145) mm, rotated rx -180 ry 0 rz 180 deg; joints [38.928, 41.405, 21.274, -137.725, 69.08, -197.984]
  Call Extruder(31613.251)
  MoveL 3377 to (-33.29, 26.54, 145) mm, rotated rx -180 ry 0 rz -180 deg; joints [38.772, 40.1, 23.738, -138.175, 69.894, -197.099]
  Call Extruder(31628.147)
  MoveL 3378 to (-38.36, 18.47, 145) mm, rotated rx 180 ry 0 rz 180 deg; joints [38.277, 38.881, 26.037, -138.935, 70.562, -196.169]
  Call Extruder(31643.042)
  MoveL 3379 to (-41.5, 9.47, 145) mm, rotated rx 180 ry 0 rz -180 deg; joints [37.447, 37.811, 28.054, -139.996, 71.057, -195.24]
  Call Extruder(31657.938)
  MoveL 3380 to (-42.57, 0, 145) mm, rotated rx 180 ry 0 rz 180 deg; joints [36.31, 36.947, 29.68, -141.322, 71.356, -194.355]
  Call Extruder(31665.493)
  MoveL 3381 to (-42.03, -4.8, 145) mm, rotated rx 180 ry 0 rz 180 deg; joints [35.612, 36.634, 30.269, -142.094, 71.402, -193.946]
  Set speed (130.0 mm/s)
  MoveL 3382 to (-54.1, -7.67, 145) mm, rotated rx 180 ry 0 rz 180 deg; joints [36.421, 35.145, 33.067, -141.53, 72.622, -193.351]
  Call Extruder(31669.565)
  Set speed (30.0 mm/s)
  MoveL 3383 to (-53.59, -12.23, 145) mm, rotated rx -180 ry 0 rz -180 deg; joints [35.732, 34.853, 33.616, -142.282, 72.667, -192.975]
  Call Extruder(31680.495)
  MoveL 3384 to (-49.53, -23.85, 145) mm, rotated rx 180 ry 0 rz -180 deg; joints [33.663, 34.433, 34.404, -144.468, 72.513, -192.112]
  Call Extruder(31691.426)
  MoveL 3385 to (-42.98, -34.27, 145) mm, rotated rx 180 ry 0 rz 180 deg; joints [31.506, 34.421, 34.427, -146.686, 72.082, -191.431]
  Call Extruder(31702.356)
  MoveL 3386 to (-34.27, -42.98, 145) mm, rotated rx 180 ry 0 rz 180 deg; joints [29.427, 34.817, 33.683, -148.773, 71.384, -190.953]
  Call Extruder(31713.286)
  MoveL 3387 to (-23.85, -49.52, 145) mm, rotated rx 180 ry 0 rz 180 deg; joints [27.581, 35.596, 32.22, -150.572, 70.447, -190.691]
  Call Extruder(31724.216)
  MoveL 3388 to (-12.23, -53.59, 145) mm, rotated rx 180 ry 0 rz 180 deg; joints [26.087, 36.709, 30.128, -151.963, 69.312, -190.655]
  Call Extruder(31735.146)
  MoveL 3389 to (0, -54.97, 145) mm, rotated rx 180 ry 0 rz -180 deg; joints [25.019, 38.089, 27.53, -152.869, 68.033, -190.85]
  Call Extruder(31741.600)
  MoveL 3390 to (7.22, -54.15, 145) mm, rotated rx 180 ry 0 rz 180 deg; joints [24.652, 39.012, 25.79, -153.106, 67.235, -191.104]
  Call Extruder(31746.077)
  MoveL 3391 to (12.23, -53.59, 145) mm, rotated rx -180 ry 0 rz -180 deg; joints [24.406, 39.66, 24.567, -153.258, 66.675, -191.282]
  Call Extruder(31757.007)
  MoveL 3392 to (23.85, -49.52, 145) mm, rotated rx -180 ry 0 rz -180 deg; joints [24.239, 41.343, 21.39, -153.137, 65.308, -191.947]
  Call Extruder(31767.937)
  MoveL 3393 to (34.27, -42.98, 145) mm, rotated rx -180 ry 0 rz -180 deg; joints [24.487, 43.055, 18.153, -152.539, 64.005, -192.832]
  Call Extruder(31778.867)
  MoveL 3394 to (42.98, -34.27, 145) mm, rotated rx -180 ry 0 rz -180 deg; joints [25.101, 44.717, 15.009, -151.523, 62.837, -193.909]
  Call Extruder(31789.797)
  MoveL 3395 to (49.52, -23.85, 145) mm, rotated rx -180 ry 0 rz 180 deg; joints [26.025, 46.252, 12.103, -150.164, 61.871, -195.131]
  Call Extruder(31800.728)
  MoveL 3396 to (53.59, -12.23, 145) mm, rotated rx 180 ry 0 rz -180 deg; joints [27.2, 47.586, 9.575, -148.546, 61.163, -196.438]
  Call Extruder(31811.658)
  MoveL 3397 to (54.97, 0, 145) mm, rotated rx 180 ry 0 rz 180 deg; joints [28.57, 48.655, 7.548, -146.764, 60.756, -197.751]
  Call Extruder(31822.588)
  MoveL 3398 to (53.59, 12.23, 145) mm, rotated rx -180 ry 0 rz 180 deg; joints [30.077, 49.405, 6.125, -144.913, 60.675, -198.986]
  Call Extruder(31833.518)
  MoveL 3399 to (49.52, 23.85, 145) mm, rotated rx 180 ry 0 rz 180 deg; joints [31.665, 49.796, 5.383, -143.083, 60.922, -200.059]
  Call Extruder(31844.448)
  MoveL 3400 to (42.98, 34.27, 145) mm, rotated rx 180 ry 0 rz 180 deg; joints [33.282, 49.807, 5.362, -141.351, 61.48, -200.899]
  Call Extruder(31855.379)
  MoveL 3401 to (34.27, 42.98, 145) mm, rotated rx 180 ry 0 rz -180 deg; joints [34.874, 49.438, 6.062, -139.78, 62.31, -201.453]
  Call Extruder(31866.309)
  MoveL 3402 to (23.85, 49.53, 145) mm, rotated rx 180 ry 0 rz -180 deg; joints [36.387, 48.708, 7.446, -138.418, 63.361, -201.694]
  Call Extruder(31877.239)
  MoveL 3403 to (12.23, 53.59, 145) mm, rotated rx 180 ry 0 rz -180 deg; joints [37.766, 47.657, 9.44, -137.301, 64.569, -201.616]
  Call Extruder(31888.169)
  MoveL 3404 to (0, 54.97, 145) mm, rotated rx -180 ry 0 rz -180 deg; joints [38.954, 46.336, 11.943, -136.455, 65.866, -201.237]
  Call Extruder(31899.099)
  MoveL 3405 to (-12.23, 53.59, 145) mm, rotated rx -180 ry 0 rz 180 deg; joints [39.895, 44.812, 14.83, -135.907, 67.185, -200.59]
  Call Extruder(31910.030)
  MoveL 3406 to (-23.85, 49.52, 145) mm, rotated rx 180 ry 0 rz 180 deg; joints [40.528, 43.155, 17.964, -135.685, 68.463, -199.719]
  Call Extruder(31920.960)
  MoveL 3407 to (-34.27, 42.98, 145) mm, rotated rx 180 ry 0 rz 180 deg; joints [40.799, 41.444, 21.2, -135.818, 69.644, -198.678]
  Call Extruder(31931.890)
  MoveL 3408 to (-42.98, 34.27, 145) mm, rotated rx 180 ry 0 rz 180 deg; joints [40.659, 39.757, 24.385, -136.335, 70.679, -197.525]
  Call Extruder(31942.820)
  MoveL 3409 to (-49.53, 23.85, 145) mm, rotated rx 180 ry 0 rz -180 deg; joints [40.072, 38.177, 27.365, -137.256, 71.528, -196.321]
  Call Extruder(31953.750)
  MoveL 3410 to (-53.59, 12.23, 145) mm, rotated rx 180 ry 0 rz 180 deg; joints [39.031, 36.783, 29.988, -138.582, 72.159, -195.124]
  Call Extruder(31964.681)
  MoveL 3411 to (-54.97, 0, 145) mm, rotated rx -180 ry 0 rz -180 deg; joints [37.56, 35.653, 32.113, -140.281, 72.545, -193.993]
  Call Extruder(31970.206)
  MoveL 3412 to (-54.27, -6.18, 145) mm, rotated rx 180 ry 0 rz -180 deg; joints [36.644, 35.242, 32.885, -141.285, 72.607, -193.474]
  Set speed (130.0 mm/s)
  MoveL 3413 to (-49.9, -9.51, 145) mm, rotated rx 180 ry 0 rz 180 deg; joints [35.741, 35.445, 32.505, -142.172, 72.259, -193.312]
  MoveL 3414 to (2.97, -12.99, 145) mm, rotated rx 180 ry 0 rz 180 deg; joints [30.614, 41.106, 21.839, -146.398, 66.955, -194.58]
  Call Extruder(31974.870)
  Set speed (80.0 mm/s)
  MoveL 3415 to (5.78, -12.01, 145) mm, rotated rx 180 ry 0 rz -180 deg; joints [30.526, 41.512, 21.072, -146.405, 66.632, -194.76]
  Call Extruder(31979.533)
  MoveL 3416 to (8.31, -10.42, 145) mm, rotated rx 180 ry 0 rz -180 deg; joints [30.538, 41.928, 20.285, -146.303, 66.327, -194.989]
  Call Extruder(31984.198)
  MoveL 3417 to (10.42, -8.31, 145) mm, rotated rx 180 ry 0 rz -180 deg; joints [30.649, 42.333, 19.519, -146.098, 66.056, -195.256]
  Call Extruder(31988.861)
  MoveL 3418 to (12.01, -5.78, 145) mm, rotated rx 180 ry 0 rz 180 deg; joints [30.85, 42.708, 18.81, -145.802, 65.833, -195.547]
  Call Extruder(31993.525)
  MoveL 3419 to (12.99, -2.97, 145) mm, rotated rx 180 ry 0 rz -180 deg; joints [31.131, 43.033, 18.195, -145.432, 65.669, -195.848]
  Call Extruder(31998.189)
  MoveL 3420 to (13.33, 0, 145) mm, rotated rx -180 ry 0 rz -180 deg; joints [31.476, 43.293, 17.703, -145.008, 65.574, -196.144]
  Call Extruder(32002.853)
  MoveL 3421 to (12.99, 2.97, 145) mm, rotated rx -180 ry 0 rz -180 deg; joints [31.869, 43.475, 17.359, -144.551, 65.552, -196.418]
  Call Extruder(32007.516)
  MoveL 3422 to (12.01, 5.78, 145) mm, rotated rx 180 ry 0 rz 180 deg; joints [32.292, 43.57, 17.18, -144.083, 65.604, -196.656]
  Call Extruder(32012.180)
  MoveL 3423 to (10.42, 8.31, 145) mm, rotated rx -180 ry 0 rz 180 deg; joints [32.725, 43.573, 17.175, -143.627, 65.726, -196.845]
  Call Extruder(32016.844)
  MoveL 3424 to (8.31, 10.42, 145) mm, rotated rx 180 ry 0 rz 180 deg; joints [33.149, 43.483, 17.344, -143.204, 65.914, -196.976]
  Call Extruder(32021.508)
  MoveL 3425 to (5.78, 12.01, 145) mm, rotated rx 180 ry 0 rz -180 deg; joints [33.544, 43.306, 17.679, -142.832, 66.155, -197.04]
  Call Extruder(32026.171)
  MoveL 3426 to (2.97, 13, 145) mm, rotated rx 180 ry 0 rz -180 deg; joints [33.893, 43.051, 18.162, -142.529, 66.439, -197.035]
  Call Extruder(32030.835)
  MoveL 3427 to (0, 13.33, 145) mm, rotated rx 180 ry 0 rz 180 deg; joints [34.177, 42.729, 18.771, -142.308, 66.749, -196.962]
  Call Extruder(32035.499)
  MoveL 3428 to (-2.97, 13, 145) mm, rotated rx 180 ry 0 rz 180 deg; joints [34.384, 42.356, 19.475, -142.18, 67.071, -196.826]
  Call Extruder(32040.163)
  MoveL 3429 to (-5.78, 12.01, 145) mm, rotated rx 180 ry 0 rz -180 deg; joints [34.5, 41.952, 20.239, -142.152, 67.389, -196.633]
  Call Extruder(32044.826)
  MoveL 3430 to (-8.31, 10.42, 145) mm, rotated rx -180 ry 0 rz 180 deg; joints [34.518, 41.536, 21.026, -142.227, 67.687, -196.395]
  Call Extruder(32049.491)
  MoveL 3431 to (-10.42, 8.31, 145) mm, rotated rx -180 ry 0 rz -180 deg; joints [34.436, 41.129, 21.795, -142.403, 67.95, -196.123]
  Call Extruder(32054.154)
  MoveL 3432 to (-12.01, 5.78, 145) mm, rotated rx 180 ry 0 rz 180 deg; joints [34.254, 40.751, 22.508, -142.673, 68.167, -195.833]
  Call Extruder(32058.818)
  MoveL 3433 to (-12.99, 2.97, 145) mm, rotated rx 180 ry 0 rz -180 deg; joints [33.981, 40.422, 23.13, -143.026, 68.326, -195.538]
  Call Extruder(32063.482)
  MoveL 3434 to (-13.33, 0, 145) mm, rotated rx 180 ry 0 rz 180 deg; joints [33.63, 40.158, 23.628, -143.447, 68.42, -195.253]
  Call Extruder(32068.146)
  MoveL 3435 to (-13, -2.97, 145) mm, rotated rx 180 ry 0 rz -180 deg; joints [33.218, 39.973, 23.977, -143.913, 68.445, -194.991]
  Call Extruder(32072.809)
  MoveL 3436 to (-12.01, -5.78, 145) mm, rotated rx -180 ry 0 rz 180 deg; joints [32.767, 39.877, 24.159, -144.401, 68.399, -194.765]
  Call Extruder(32077.473)
  MoveL 3437 to (-10.42, -8.31, 145) mm, rotated rx 180 ry 0 rz -180 deg; joints [32.302, 39.874, 24.164, -144.885, 68.283, -194.585]
  Call Extruder(32082.137)
  MoveL 3438 to (-8.31, -10.42, 145) mm, rotated rx 180 ry 0 rz 180 deg; joints [31.85, 39.965, 23.992, -145.338, 68.103, -194.459]
  Call Extruder(32086.801)
  MoveL 3439 to (-5.78, -12.01, 145) mm, rotated rx 180 ry 0 rz -180 deg; joints [31.435, 40.145, 23.653, -145.735, 67.868, -194.394]
  Call Extruder(32091.464)
  MoveL 3440 to (-2.97, -12.99, 145) mm, rotated rx 180 ry 0 rz -180 deg; joints [31.079, 40.404, 23.163, -146.055, 67.589, -194.393]
  Call Extruder(32096.128)
  MoveL 3441 to (0, -13.33, 145) mm, rotated rx 180 ry 0 rz 180 deg; joints [30.801, 40.73, 22.548, -146.279, 67.28, -194.455]
  Call Extruder(32100.792)
  MoveL 3442 to (2.97, -12.99, 145) mm, rotated rx 180 ry 0 rz 180 deg; joints [30.614, 41.106, 21.839, -146.398, 66.955, -194.58]
  Set speed (130.0 mm/s)
  MoveL 3443 to (2.97, -12.99, 150) mm, rotated rx 180 ry 0 rz 180 deg; joints [30.614, 40.289, 21.947, -146.228, 66.365, -195.008]
  MoveL 3444 to (-26.25, -4.54, 150) mm, rotated rx 180 ry 0 rz -180 deg; joints [34.172, 37.506, 27.116, -143.079, 69.231, -194.92]
  Call Extruder(32103.025)
  Set speed (60.0 mm/s)
  MoveL 3445 to (-26.09, -5.96, 150) mm, rotated rx 180 ry 0 rz 180 deg; joints [33.969, 37.416, 27.283, -143.306, 69.241, -194.796]
  Call Extruder(32112.390)
  MoveL 3446 to (-24.12, -11.61, 150) mm, rotated rx -180 ry 0 rz 180 deg; joints [33.033, 37.216, 27.653, -144.313, 69.143, -194.344]
  Call Extruder(32121.754)
  MoveL 3447 to (-20.93, -16.69, 150) mm, rotated rx 180 ry 0 rz -180 deg; joints [32.066, 37.21, 27.664, -145.319, 68.91, -193.981]
  Call Extruder(32131.120)
  MoveL 3448 to (-16.69, -20.93, 150) mm, rotated rx -180 ry 0 rz 180 deg; joints [31.126, 37.399, 27.315, -146.263, 68.552, -193.723]
  Call Extruder(32140.485)
  MoveL 3449 to (-11.61, -24.11, 150) mm, rotated rx 180 ry 0 rz -180 deg; joints [30.272, 37.771, 26.625, -147.087, 68.085, -193.581]
  Call Extruder(32149.849)
  MoveL 3450 to (-5.96, -26.09, 150) mm, rotated rx 180 ry 0 rz -180 deg; joints [29.552, 38.307, 25.631, -147.742, 67.53, -193.562]
  Call Extruder(32159.214)
  MoveL 3451 to (0, -26.77, 150) mm, rotated rx 180 ry 0 rz -180 deg; joints [29.003, 38.977, 24.387, -148.193, 66.914, -193.668]
  Call Extruder(32168.580)
  MoveL 3452 to (5.96, -26.09, 150) mm, rotated rx -180 ry 0 rz -180 deg; joints [28.65, 39.746, 22.957, -148.416, 66.268, -193.898]
  Call Extruder(32177.944)
  MoveL 3453 to (11.61, -24.11, 150) mm, rotated rx 180 ry 0 rz -180 deg; joints [28.503, 40.575, 21.413, -148.406, 65.624, -194.244]
  Call Extruder(32187.309)
  MoveL 3454 to (16.69, -20.93, 150) mm, rotated rx 180 ry 0 rz 180 deg; joints [28.559, 41.422, 19.834, -148.168, 65.016, -194.692]
  Call Extruder(32196.675)
  MoveL 3455 to (20.93, -16.69, 150) mm, rotated rx 180 ry 0 rz -180 deg; joints [28.808, 42.246, 18.298, -147.724, 64.475, -195.224]
  Call Extruder(32206.039)
  MoveL 3456 to (24.12, -11.61, 150) mm, rotated rx 180 ry 0 rz -180 deg; joints [29.229, 43.006, 16.879, -147.103, 64.033, -195.814]
  Call Extruder(32215.404)
  MoveL 3457 to (26.09, -5.96, 150) mm, rotated rx -180 ry 0 rz -180 deg; joints [29.796, 43.665, 15.647, -146.341, 63.711, -196.431]
  Call Extruder(32224.769)
  MoveL 3458 to (26.77, 0, 150) mm, rotated rx -180 ry 0 rz -180 deg; joints [30.482, 44.192, 14.662, -145.482, 63.529, -197.044]
  Call Extruder(32234.134)
  MoveL 3459 to (26.09, 5.96, 150) mm, rotated rx 180 ry 0 rz 180 deg; joints [31.252, 44.559, 13.973, -144.568, 63.496, -197.616]
  Call Extruder(32243.499)
  MoveL 3460 to (24.11, 11.61, 150) mm, rotated rx 180 ry 0 rz -180 deg; joints [32.076, 44.751, 13.615, -143.644, 63.613, -198.115]
  Call Extruder(32252.864)
  MoveL 3461 to (20.93, 16.69, 150) mm, rotated rx 180 ry 0 rz -180 deg; joints [32.917, 44.757, 13.605, -142.752, 63.874, -198.512]
  Call Extruder(32262.229)
  MoveL 3462 to (16.69, 20.93, 150) mm, rotated rx 180 ry 0 rz 180 deg; joints [33.742, 44.576, 13.943, -141.929, 64.263, -198.785]
  Call Extruder(32271.594)
  MoveL 3463 to (11.61, 24.12, 150) mm, rotated rx 180 ry 0 rz -180 deg; joints [34.517, 44.218, 14.613, -141.209, 64.757, -198.92]
  Call Extruder(32280.959)
  MoveL 3464 to (5.96, 26.09, 150) mm, rotated rx 180 ry 0 rz -180 deg; joints [35.208, 43.7, 15.581, -140.62, 65.331, -198.911]
  Call Extruder(32290.324)
  MoveL 3465 to (0, 26.77, 150) mm, rotated rx -180 ry 0 rz -180 deg; joints [35.784, 43.048, 16.8, -140.186, 65.954, -198.761]
  Call Extruder(32299.689)
  MoveL 3466 to (-5.96, 26.09, 150) mm, rotated rx 180 ry 0 rz -180 deg; joints [36.214, 42.293, 18.21, -139.926, 66.593, -198.48]
  Call Extruder(32309.054)
  MoveL 3467 to (-11.61, 24.12, 150) mm, rotated rx 180 ry 0 rz 180 deg; joints [36.473, 41.472, 19.742, -139.853, 67.218, -198.088]
  Call Extruder(32318.419)
  MoveL 3468 to (-16.69, 20.93, 150) mm, rotated rx 180 ry 0 rz -180 deg; joints [36.542, 40.625, 21.321, -139.978, 67.799, -197.605]
  Call Extruder(32327.784)
  MoveL 3469 to (-20.93, 16.69, 150) mm, rotated rx 180 ry 0 rz -180 deg; joints [36.407, 39.794, 22.868, -140.302, 68.308, -197.058]
  Call Extruder(32337.149)
  MoveL 3470 to (-24.12, 11.61, 150) mm, rotated rx 180 ry 0 rz 180 deg; joints [36.065, 39.02, 24.307, -140.819, 68.724, -196.475]
  Call Extruder(32346.514)
  MoveL 3471 to (-26.09, 5.96, 150) mm, rotated rx -180 ry 0 rz -180 deg; joints [35.528, 38.343, 25.564, -141.513, 69.026, -195.886]
  Call Extruder(32355.879)
  MoveL 3472 to (-26.77, 0, 150) mm, rotated rx 180 ry 0 rz 180 deg; joints [34.817, 37.798, 26.574, -142.356, 69.201, -195.317]
  Call Extruder(32360.668)
  MoveL 3473 to (-26.42, -3.05, 150) mm, rotated rx 180 ry 0 rz -180 deg; joints [34.385, 37.601, 26.94, -142.84, 69.221, -195.05]
  Set speed (130.0 mm/s)
  MoveL 3474 to (-41.86, -6.29, 150) mm, rotated rx 180 ry 0 rz -180 deg; joints [35.393, 35.644, 30.56, -142.171, 70.797, -194.327]
  Call Extruder(32365.666)
  Set speed (60.0 mm/s)
  MoveL 3475 to (-41.5, -9.47, 150) mm, rotated rx -180 ry 0 rz 180 deg; joints [34.924, 35.439, 30.938, -142.689, 70.819, -194.057]
  Call Extruder(32380.561)
  MoveL 3476 to (-38.36, -18.47, 150) mm, rotated rx -180 ry 0 rz 180 deg; joints [33.373, 35.114, 31.539, -144.342, 70.673, -193.357]
  Call Extruder(32395.457)
  MoveL 3477 to (-33.28, -26.54, 150) mm, rotated rx -180 ry 0 rz 180 deg; joints [31.763, 35.104, 31.556, -146.008, 70.315, -192.797]
  Call Extruder(32410.353)
  MoveL 3478 to (-26.54, -33.29, 150) mm, rotated rx -180 ry 0 rz 180 deg; joints [30.206, 35.411, 30.99, -147.573, 69.758, -192.396]
  Call Extruder(32425.249)
  MoveL 3479 to (-18.47, -38.36, 150) mm, rotated rx 180 ry 0 rz -180 deg; joints [28.808, 36.016, 29.873, -148.932, 69.026, -192.17]
  Call Extruder(32440.144)
  MoveL 3480 to (-9.47, -41.5, 150) mm, rotated rx 180 ry 0 rz -180 deg; joints [27.654, 36.882, 28.271, -149.996, 68.149, -192.129]
  Call Extruder(32455.040)
  MoveL 3481 to (0, -42.57, 150) mm, rotated rx 180 ry 0 rz -180 deg; joints [26.805, 37.96, 26.274, -150.707, 67.171, -192.28]
  Call Extruder(32469.936)
  MoveL 3482 to (9.47, -41.5, 150) mm, rotated rx 180 ry 0 rz 180 deg; joints [26.29, 39.191, 23.988, -151.033, 66.138, -192.622]
  Call Extruder(32484.832)
  MoveL 3483 to (18.47, -38.36, 150) mm, rotated rx 180 ry 0 rz 180 deg; joints [26.114, 40.513, 21.529, -150.971, 65.104, -193.15]
  Call Extruder(32499.728)
  MoveL 3484 to (26.54, -33.28, 150) mm, rotated rx 180 ry 0 rz -180 deg; joints [26.262, 41.859, 19.019, -150.542, 64.124, -193.847]
  Call Extruder(32514.624)
  MoveL 3485 to (33.28, -26.54, 150) mm, rotated rx 180 ry 0 rz 180 deg; joints [26.703, 43.166, 16.58, -149.786, 63.25, -194.687]
  Call Extruder(32529.519)
  MoveL 3486 to (38.36, -18.47, 150) mm, rotated rx 180 ry 0 rz -180 deg; joints [27.4, 44.37, 14.328, -148.757, 62.531, -195.633]
  Call Extruder(32544.415)
  MoveL 3487 to (41.5, -9.47, 150) mm, rotated rx 180 ry 0 rz -180 deg; joints [28.309, 45.415, 12.371, -147.518, 62.009, -196.636]
  Call Extruder(32559.311)
  MoveL 3488 to (42.57, 0, 150) mm, rotated rx 180 ry 0 rz -180 deg; joints [29.382, 46.251, 10.805, -146.14, 61.715, -197.638]
  Call Extruder(32574.207)
  MoveL 3489 to (41.51, 9.47, 150) mm, rotated rx -180 ry 0 rz -180 deg; joints [30.575, 46.835, 9.709, -144.696, 61.664, -198.578]
  Call Extruder(32589.102)
  MoveL 3490 to (38.36, 18.47, 150) mm, rotated rx 180 ry 0 rz -180 deg; joints [31.839, 47.14, 9.138, -143.255, 61.86, -199.398]
  Call Extruder(32603.998)
  MoveL 3491 to (33.28, 26.54, 150) mm, rotated rx -180 ry 0 rz -180 deg; joints [33.128, 47.149, 9.121, -141.88, 62.288, -200.046]
  Call Extruder(32618.894)
  MoveL 3492 to (26.54, 33.29, 150) mm, rotated rx 180 ry 0 rz -180 deg; joints [34.394, 46.861, 9.66, -140.623, 62.924, -200.485]
  Call Extruder(32633.790)
  MoveL 3493 to (18.47, 38.36, 150) mm, rotated rx 180 ry 0 rz 180 deg; joints [35.592, 46.293, 10.727, -139.529, 63.727, -200.691]
  Call Extruder(32648.686)
  MoveL 3494 to (9.47, 41.51, 150) mm, rotated rx 180 ry 0 rz 180 deg; joints [36.675, 45.471, 12.267, -138.631, 64.651, -200.658]
  Call Extruder(32663.581)
  MoveL 3495 to (0, 42.57, 150) mm, rotated rx -180 ry 0 rz -180 deg; joints [37.594, 44.437, 14.203, -137.96, 65.647, -200.395]
  Call Extruder(32678.477)
  MoveL 3496 to (-9.47, 41.5, 150) mm, rotated rx 180 ry 0 rz 180 deg; joints [38.304, 43.24, 16.441, -137.541, 66.663, -199.924]
  Call Extruder(32693.373)
  MoveL 3497 to (-18.47, 38.36, 150) mm, rotated rx 180 ry 0 rz -180 deg; joints [38.762, 41.938, 18.873, -137.394, 67.649, -199.278]
  Call Extruder(32708.269)
  MoveL 3498 to (-26.54, 33.29, 150) mm, rotated rx 180 ry 0 rz -180 deg; joints [38.928, 40.592, 21.381, -137.541, 68.56, -198.494]
  Call Extruder(32723.165)
  MoveL 3499 to (-33.29, 26.54, 150) mm, rotated rx 180 ry 0 rz 180 deg; joints [38.772, 39.267, 23.846, -137.995, 69.355, -197.615]
  Call Extruder(32738.061)
  MoveL 3500 to (-38.36, 18.47, 150) mm, rotated rx -180 ry 0 rz 180 deg; joints [38.277, 38.029, 26.147, -138.76, 70.003, -196.688]
  Call Extruder(32752.956)
  MoveL 3501 to (-41.5, 9.47, 150) mm, rotated rx 180 ry 0 rz -180 deg; joints [37.447, 36.94, 28.164, -139.825, 70.475, -195.758]
  Call Extruder(32767.852)
  MoveL 3502 to (-42.57, 0, 150) mm, rotated rx -180 ry 0 rz 180 deg; joints [36.31, 36.06, 29.792, -141.155, 70.752, -194.868]
  Call Extruder(32775.406)
  MoveL 3503 to (-42.03, -4.8, 150) mm, rotated rx 180 ry 0 rz -180 deg; joints [35.612, 35.741, 30.381, -141.929, 70.786, -194.455]
  Set speed (130.0 mm/s)
  MoveL 3504 to (-54.1, -7.67, 150) mm, rotated rx 180 ry 0 rz -180 deg; joints [36.421, 34.222, 33.181, -141.369, 71.989, -193.88]
  Call Extruder(32779.479)
  Set speed (30.0 mm/s)
  MoveL 3505 to (-53.59, -12.23, 150) mm, rotated rx 180 ry 0 rz 180 deg; joints [35.732, 33.924, 33.73, -142.123, 72.023, -193.499]
  Call Extruder(32790.409)
  MoveL 3506 to (-49.53, -23.85, 150) mm, rotated rx 180 ry 0 rz -180 deg; joints [33.663, 33.495, 34.519, -144.314, 71.844, -192.615]
  Call Extruder(32801.339)
  MoveL 3507 to (-42.98, -34.27, 150) mm, rotated rx 180 ry 0 rz -180 deg; joints [31.506, 33.483, 34.541, -146.537, 71.394, -191.908]
  Call Extruder(32812.269)
  MoveL 3508 to (-34.27, -42.98, 150) mm, rotated rx 180 ry 0 rz -180 deg; joints [29.427, 33.888, 33.797, -148.627, 70.687, -191.401]
  Call Extruder(32823.200)
  MoveL 3509 to (-23.85, -49.52, 150) mm, rotated rx 180 ry 0 rz -180 deg; joints [27.581, 34.683, 32.333, -150.429, 69.751, -191.11]
  Call Extruder(32834.130)
  MoveL 3510 to (-12.23, -53.59, 150) mm, rotated rx 180 ry 0 rz -180 deg; joints [26.087, 35.817, 30.24, -151.822, 68.624, -191.048]
  Call Extruder(32845.060)
  MoveL 3511 to (0, -54.97, 150) mm, rotated rx 180 ry 0 rz 180 deg; joints [25.019, 37.223, 27.641, -152.728, 67.361, -191.224]
  Call Extruder(32855.558)
  MoveL 3512 to (11.75, -53.65, 150) mm, rotated rx 180 ry 0 rz 180 deg; joints [24.429, 38.757, 24.795, -153.1, 66.077, -191.625]
  Call Extruder(32855.990)
  MoveL 3513 to (12.23, -53.59, 150) mm, rotated rx -180 ry 0 rz -180 deg; joints [24.406, 38.821, 24.676, -153.114, 66.023, -191.642]
  Call Extruder(32866.921)
  MoveL 3514 to (23.85, -49.52, 150) mm, rotated rx 180 ry 0 rz -180 deg; joints [24.239, 40.53, 21.498, -152.987, 64.679, -192.3]
  Call Extruder(32877.851)
  MoveL 3515 to (34.27, -42.98, 150) mm, rotated rx 180 ry 0 rz 180 deg; joints [24.487, 42.266, 18.261, -152.383, 63.4, -193.184]
  Call Extruder(32888.781)
  MoveL 3516 to (42.98, -34.27, 150) mm, rotated rx -180 ry 0 rz -180 deg; joints [25.101, 43.949, 15.115, -151.359, 62.256, -194.265]
  Call Extruder(32899.711)
  MoveL 3517 to (49.52, -23.85, 150) mm, rotated rx 180 ry 0 rz 180 deg; joints [26.025, 45.501, 12.21, -149.99, 61.313, -195.496]
  Call Extruder(32910.641)
  MoveL 3518 to (53.59, -12.23, 150) mm, rotated rx 180 ry 0 rz -180 deg; joints [27.2, 46.85, 9.682, -148.363, 60.627, -196.814]
  Call Extruder(32921.572)
  MoveL 3519 to (54.97, 0, 150) mm, rotated rx 180 ry 0 rz -180 deg; joints [28.57, 47.93, 7.655, -146.572, 60.24, -198.141]
  Call Extruder(32932.502)
  MoveL 3520 to (53.59, 12.23, 150) mm, rotated rx -180 ry 0 rz -180 deg; joints [30.077, 48.687, 6.233, -144.714, 60.176, -199.39]
  Call Extruder(32943.432)
  MoveL 3521 to (49.52, 23.85, 150) mm, rotated rx 180 ry 0 rz -180 deg; joints [31.665, 49.082, 5.491, -142.878, 60.438, -200.477]
  Call Extruder(32954.362)
  MoveL 3522 to (42.98, 34.27, 150) mm, rotated rx 180 ry 0 rz -180 deg; joints [33.282, 49.093, 5.47, -141.142, 61.007, -201.331]
  Call Extruder(32965.292)
  MoveL 3523 to (34.27, 42.98, 150) mm, rotated rx 180 ry 0 rz 180 deg; joints [34.874, 48.721, 6.17, -139.571, 61.846, -201.9]
  Call Extruder(32976.223)
  MoveL 3524 to (23.85, 49.53, 150) mm, rotated rx 180 ry 0 rz -180 deg; joints [36.387, 47.984, 7.553, -138.211, 62.9, -202.154]
  Call Extruder(32987.153)
  MoveL 3525 to (12.23, 53.59, 150) mm, rotated rx 180 ry 0 rz -180 deg; joints [37.766, 46.922, 9.547, -137.096, 64.108, -202.089]
  Call Extruder(32998.083)
  MoveL 3526 to (0, 54.97, 150) mm, rotated rx -180 ry 0 rz 180 deg; joints [38.954, 45.587, 12.049, -136.254, 65.401, -201.724]
  Call Extruder(33009.013)
  MoveL 3527 to (-12.23, 53.59, 150) mm, rotated rx 180 ry 0 rz 180 deg; joints [39.895, 44.045, 14.936, -135.711, 66.711, -201.09]
  Call Extruder(33019.943)
  MoveL 3528 to (-23.85, 49.53, 150) mm, rotated rx 180 ry 0 rz 180 deg; joints [40.528, 42.367, 18.071, -135.495, 67.976, -200.232]
  Call Extruder(33030.874)
  MoveL 3529 to (-34.27, 42.98, 150) mm, rotated rx 180 ry 0 rz -180 deg; joints [40.799, 40.632, 21.308, -135.633, 69.139, -199.204]
  Call Extruder(33041.804)
  MoveL 3530 to (-42.98, 34.27, 150) mm, rotated rx 180 ry 0 rz -180 deg; joints [40.659, 38.919, 24.494, -136.156, 70.152, -198.061]
  Call Extruder(33052.734)
  MoveL 3531 to (-49.53, 23.85, 150) mm, rotated rx -180 ry 0 rz -180 deg; joints [40.072, 37.312, 27.475, -137.082, 70.975, -196.862]
  Call Extruder(33063.664)
  MoveL 3532 to (-53.59, 12.23, 150) mm, rotated rx -180 ry 0 rz -180 deg; joints [39.031, 35.893, 30.1, -138.413, 71.576, -195.667]
  Call Extruder(33074.594)
  MoveL 3533 to (-54.97, 0, 150) mm, rotated rx 180 ry 0 rz 180 deg; joints [37.56, 34.741, 32.226, -140.117, 71.931, -194.53]
  Call Extruder(33080.120)
  MoveL 3534 to (-54.27, -6.18, 150) mm, rotated rx 180 ry 0 rz 180 deg; joints [36.644, 34.322, 32.998, -141.124, 71.978, -194.005]
  Set speed (130.0 mm/s)
  MoveL 3535 to (-49.9, -9.51, 150) mm, rotated rx 180 ry 0 rz 180 deg; joints [35.741, 34.528, 32.618, -142.011, 71.625, -193.831]
  MoveL 3536 to (-4.92, 13.82, 150) mm, rotated rx 180 ry 0 rz -180 deg; joints [34.648, 41.395, 19.886, -141.76, 66.715, -197.303]
  Call Extruder(33113.295)
  Set speed (20.0 mm/s)
  MoveL 3537 to (-13.82, 4.92, 150) mm, rotated rx 180 ry 0 rz 180 deg; joints [34.301, 39.652, 23.131, -142.508, 67.801, -196.163]
  Call Extruder(33183.102)
  MoveL 3538 to (4.92, -13.82, 150) mm, rotated rx 180 ry 0 rz -180 deg; joints [30.357, 40.466, 21.616, -146.463, 66.171, -194.991]
  Call Extruder(33216.277)
  MoveL 3539 to (13.82, -4.91, 150) mm, rotated rx -180 ry 0 rz -180 deg; joints [30.824, 42.201, 18.382, -145.589, 65.053, -196.115]
  Set speed (130.0 mm/s)
  MoveL 3540 to (13.82, -4.91, 155) mm, rotated rx 180 ry 0 rz -180 deg; joints [30.824, 41.419, 18.472, -145.404, 64.483, -196.548]
  MoveL 3541 to (-26.25, -4.54, 155) mm, rotated rx 180 ry 0 rz -180 deg; joints [34.172, 36.653, 27.209, -142.902, 68.624, -195.41]
  Call Extruder(33218.509)
  Set speed (60.0 mm/s)
  MoveL 3542 to (-26.09, -5.96, 155) mm, rotated rx 180 ry 0 rz -180 deg; joints [33.969, 36.562, 27.376, -143.13, 68.631, -195.285]
  Call Extruder(33227.874)
  MoveL 3543 to (-24.12, -11.61, 155) mm, rotated rx 180 ry 0 rz 180 deg; joints [33.033, 36.358, 27.746, -144.14, 68.522, -194.824]
  Call Extruder(33237.239)
  MoveL 3544 to (-20.93, -16.69, 155) mm, rotated rx 180 ry 0 rz -180 deg; joints [32.066, 36.352, 27.756, -145.148, 68.282, -194.45]
  Call Extruder(33246.604)
  MoveL 3545 to (-16.69, -20.93, 155) mm, rotated rx -180 ry 0 rz -180 deg; joints [31.126, 36.544, 27.407, -146.093, 67.919, -194.18]
  Call Extruder(33255.969)
  MoveL 3546 to (-11.61, -24.12, 155) mm, rotated rx -180 ry 0 rz 180 deg; joints [30.272, 36.923, 26.717, -146.919, 67.451, -194.026]
  Call Extruder(33265.334)
  MoveL 3547 to (-5.96, -26.09, 155) mm, rotated rx 180 ry 0 rz -180 deg; joints [29.552, 37.467, 25.723, -147.574, 66.899, -193.995]
  Call Extruder(33274.699)
  MoveL 3548 to (0, -26.77, 155) mm, rotated rx -180 ry 0 rz -180 deg; joints [29.003, 38.148, 24.478, -148.024, 66.289, -194.092]
  Call Extruder(33284.064)
  MoveL 3549 to (5.96, -26.09, 155) mm, rotated rx 180 ry 0 rz 180 deg; joints [28.65, 38.929, 23.047, -148.246, 65.65, -194.315]
  Call Extruder(33293.429)
  MoveL 3550 to (11.61, -24.11, 155) mm, rotated rx 180 ry 0 rz 180 deg; joints [28.503, 39.771, 21.504, -148.233, 65.016, -194.656]
  Call Extruder(33302.794)
  MoveL 3551 to (16.69, -20.93, 155) mm, rotated rx 180 ry 0 rz -180 deg; joints [28.559, 40.63, 19.925, -147.993, 64.42, -195.103]
  Call Extruder(33312.159)
  MoveL 3552 to (20.93, -16.69, 155) mm, rotated rx 180 ry 0 rz -180 deg; joints [28.808, 41.465, 18.388, -147.545, 63.892, -195.635]
  Call Extruder(33321.524)
  MoveL 3553 to (24.12, -11.61, 155) mm, rotated rx 180 ry 0 rz 180 deg; joints [29.229, 42.235, 16.968, -146.92, 63.461, -196.228]
  Call Extruder(33330.889)
  MoveL 3554 to (26.09, -5.96, 155) mm, rotated rx 180 ry 0 rz 180 deg; joints [29.796, 42.902, 15.736, -146.154, 63.151, -196.85]
  Call Extruder(33340.254)
  MoveL 3555 to (26.77, 0, 155) mm, rotated rx 180 ry 0 rz -180 deg; joints [30.482, 43.435, 14.751, -145.291, 62.98, -197.468]
  Call Extruder(33349.619)
  MoveL 3556 to (26.09, 5.96, 155) mm, rotated rx 180 ry 0 rz 180 deg; joints [31.252, 43.807, 14.063, -144.373, 62.957, -198.047]
  Call Extruder(33358.984)
  MoveL 3557 to (24.11, 11.61, 155) mm, rotated rx 180 ry 0 rz -180 deg; joints [32.076, 44.001, 13.705, -143.447, 63.082, -198.554]
  Call Extruder(33368.349)
  MoveL 3558 to (20.93, 16.69, 155) mm, rotated rx 180 ry 0 rz -180 deg; joints [32.917, 44.006, 13.694, -142.553, 63.349, -198.959]
  Call Extruder(33377.714)
  MoveL 3559 to (16.69, 20.93, 155) mm, rotated rx 180 ry 0 rz 180 deg; joints [33.742, 43.824, 14.032, -141.73, 63.742, -199.241]
  Call Extruder(33387.079)
  MoveL 3560 to (11.61, 24.12, 155) mm, rotated rx -180 ry 0 rz -180 deg; joints [34.517, 43.461, 14.702, -141.009, 64.238, -199.384]
  Call Extruder(33396.444)
  MoveL 3561 to (5.96, 26.09, 155) mm, rotated rx 180 ry 0 rz -180 deg; joints [35.208, 42.937, 15.671, -140.421, 64.812, -199.383]
  Call Extruder(33405.809)
  MoveL 3562 to (0, 26.77, 155) mm, rotated rx 180 ry 0 rz 180 deg; joints [35.784, 42.277, 16.89, -139.989, 65.431, -199.24]
  Call Extruder(33415.174)
  MoveL 3563 to (-5.96, 26.09, 155) mm, rotated rx 180 ry 0 rz -180 deg; joints [36.214, 41.512, 18.3, -139.73, 66.066, -198.967]
  Call Extruder(33424.539)
  MoveL 3564 to (-11.61, 24.12, 155) mm, rotated rx 180 ry 0 rz 180 deg; joints [36.473, 40.68, 19.832, -139.66, 66.683, -198.58]
  Call Extruder(33433.903)
  MoveL 3565 to (-16.69, 20.93, 155) mm, rotated rx 180 ry 0 rz 180 deg; joints [36.542, 39.821, 21.411, -139.788, 67.254, -198.102]
  Call Extruder(33443.269)
  MoveL 3566 to (-20.93, 16.69, 155) mm, rotated rx -180 ry 0 rz 180 deg; joints [36.407, 38.978, 22.959, -140.115, 67.751, -197.558]
  Call Extruder(33452.634)
  MoveL 3567 to (-24.12, 11.61, 155) mm, rotated rx 180 ry 0 rz -180 deg; joints [36.065, 38.192, 24.398, -140.635, 68.153, -196.977]
  Call Extruder(33461.998)
  MoveL 3568 to (-26.09, 5.96, 155) mm, rotated rx 180 ry 0 rz 180 deg; joints [35.528, 37.504, 25.656, -141.332, 68.442, -196.386]
  Call Extruder(33471.363)
  MoveL 3569 to (-26.77, 0, 155) mm, rotated rx -180 ry 0 rz 180 deg; joints [34.817, 36.951, 26.666, -142.177, 68.603, -195.813]
  Call Extruder(33476.152)
  MoveL 3570 to (-26.42, -3.05, 155) mm, rotated rx 180 ry 0 rz 180 deg; joints [34.385, 36.75, 27.032, -142.663, 68.618, -195.542]
  Set speed (130.0 mm/s)
  MoveL 3571 to (-41.86, -6.3, 155) mm, rotated rx 180 ry 0 rz 180 deg; joints [35.393, 34.758, 30.654, -141.998, 70.172, -194.843]
  Call Extruder(33481.150)
  Set speed (60.0 mm/s)
  MoveL 3572 to (-41.5, -9.47, 155) mm, rotated rx 180 ry 0 rz -180 deg; joints [34.924, 34.549, 31.033, -142.518, 70.187, -194.569]
  Call Extruder(33496.046)
  MoveL 3573 to (-38.36, -18.47, 155) mm, rotated rx 180 ry 0 rz 180 deg; joints [33.373, 34.218, 31.633, -144.175, 70.022, -193.855]
  Call Extruder(33510.942)
  MoveL 3574 to (-33.28, -26.54, 155) mm, rotated rx 180 ry 0 rz 180 deg; joints [31.763, 34.208, 31.65, -145.844, 69.651, -193.275]
  Call Extruder(33525.837)
  MoveL 3575 to (-26.54, -33.28, 155) mm, rotated rx -180 ry 0 rz -180 deg; joints [30.206, 34.521, 31.084, -147.412, 69.087, -192.853]
  Call Extruder(33540.733)
  MoveL 3576 to (-18.47, -38.36, 155) mm, rotated rx 180 ry 0 rz -180 deg; joints [28.808, 35.137, 29.967, -148.773, 68.354, -192.606]
  Call Extruder(33555.629)
  MoveL 3577 to (-9.47, -41.5, 155) mm, rotated rx 180 ry 0 rz -180 deg; joints [27.654, 36.019, 28.364, -149.839, 67.483, -192.546]
  Call Extruder(33570.525)
  MoveL 3578 to (0, -42.57, 155) mm, rotated rx 180 ry 0 rz -180 deg; joints [26.805, 37.115, 26.366, -150.549, 66.515, -192.682]
  Call Extruder(33585.421)
  MoveL 3579 to (9.47, -41.5, 155) mm, rotated rx 180 ry 0 rz -180 deg; joints [26.29, 38.366, 24.079, -150.873, 65.497, -193.013]
  Call Extruder(33600.316)
  MoveL 3580 to (18.47, -38.36, 155) mm, rotated rx 180 ry 0 rz 180 deg; joints [26.114, 39.708, 21.619, -150.808, 64.48, -193.534]
  Call Extruder(33615.212)
  MoveL 3581 to (26.54, -33.29, 155) mm, rotated rx 180 ry 0 rz 180 deg; joints [26.262, 41.073, 19.109, -150.374, 63.518, -194.23]
  Call Extruder(33630.108)
  MoveL 3582 to (33.28, -26.54, 155) mm, rotated rx 180 ry 0 rz 180 deg; joints [26.703, 42.397, 16.67, -149.611, 62.663, -195.072]
  Call Extruder(33645.004)
  MoveL 3583 to (38.36, -18.47, 155) mm, rotated rx -180 ry 0 rz -180 deg; joints [27.4, 43.616, 14.417, -148.575, 61.963, -196.024]
  Call Extruder(33659.899)
  MoveL 3584 to (41.5, -9.47, 155) mm, rotated rx 180 ry 0 rz -180 deg; joints [28.309, 44.673, 12.461, -147.329, 61.459, -197.035]
  Call Extruder(33674.795)
  MoveL 3585 to (42.57, 0, 155) mm, rotated rx 180 ry 0 rz 180 deg; joints [29.382, 45.517, 10.895, -145.945, 61.181, -198.047]
  Call Extruder(33689.691)
  MoveL 3586 to (41.5, 9.47, 155) mm, rotated rx -180 ry 0 rz -180 deg; joints [30.575, 46.108, 9.799, -144.495, 61.144, -198.999]
  Call Extruder(33704.587)
  MoveL 3587 to (38.36, 18.47, 155) mm, rotated rx 180 ry 0 rz 180 deg; joints [31.839, 46.416, 9.228, -143.05, 61.352, -199.83]
  Call Extruder(33719.483)
  MoveL 3588 to (33.28, 26.54, 155) mm, rotated rx 180 ry 0 rz -180 deg; joints [33.128, 46.425, 9.211, -141.672, 61.79, -200.491]
  Call Extruder(33734.379)
  MoveL 3589 to (26.54, 33.29, 155) mm, rotated rx 180 ry 0 rz 180 deg; joints [34.394, 46.134, 9.75, -140.414, 62.432, -200.941]
  Call Extruder(33749.274)
  MoveL 3590 to (18.47, 38.36, 155) mm, rotated rx 180 ry 0 rz -180 deg; joints [35.592, 45.56, 10.817, -139.32, 63.238, -201.158]
  Call Extruder(33764.170)
  MoveL 3591 to (9.47, 41.51, 155) mm, rotated rx 180 ry 0 rz 180 deg; joints [36.675, 44.729, 12.357, -138.425, 64.163, -201.137]
  Call Extruder(33779.066)
  MoveL 3592 to (0, 42.57, 155) mm, rotated rx 180 ry 0 rz -180 deg; joints [37.594, 43.683, 14.293, -137.756, 65.155, -200.885]
  Call Extruder(33793.962)
  MoveL 3593 to (-9.47, 41.51, 155) mm, rotated rx 180 ry 0 rz -180 deg; joints [38.304, 42.472, 16.531, -137.34, 66.163, -200.425]
  Call Extruder(33808.857)
  MoveL 3594 to (-18.47, 38.36, 155) mm, rotated rx -180 ry 0 rz 180 deg; joints [38.762, 41.153, 18.963, -137.198, 67.138, -199.789]
  Call Extruder(33823.753)
  MoveL 3595 to (-26.54, 33.28, 155) mm, rotated rx 180 ry 0 rz 180 deg; joints [38.928, 39.788, 21.472, -137.349, 68.034, -199.013]
  Call Extruder(33838.649)
  MoveL 3596 to (-33.29, 26.54, 155) mm, rotated rx 180 ry 0 rz -180 deg; joints [38.772, 38.444, 23.938, -137.807, 68.812, -198.141]
  Call Extruder(33853.545)
  MoveL 3597 to (-38.36, 18.47, 155) mm, rotated rx 180 ry 0 rz 180 deg; joints [38.277, 37.185, 26.238, -138.577, 69.438, -197.218]
  Call Extruder(33868.441)
  MoveL 3598 to (-41.5, 9.47, 155) mm, rotated rx 180 ry 0 rz -180 deg; joints [37.447, 36.078, 28.257, -139.646, 69.888, -196.287]
  Call Extruder(33883.336)
  MoveL 3599 to (-42.57, 0, 155) mm, rotated rx 180 ry 0 rz 180 deg; joints [36.31, 35.182, 29.885, -140.98, 70.141, -195.391]
  Call Extruder(33890.891)
  MoveL 3600 to (-42.03, -4.8, 155) mm, rotated rx 180 ry 0 rz -180 deg; joints [35.612, 34.857, 30.474, -141.756, 70.165, -194.973]
  Set speed (130.0 mm/s)
  MoveL 3601 to (-54.1, -7.67, 155) mm, rotated rx -180 ry 0 rz 180 deg; joints [36.421, 33.309, 33.276, -141.199, 71.351, -194.419]
  Call Extruder(33894.963)
  Set speed (30.0 mm/s)
  MoveL 3602 to (-53.59, -12.23, 155) mm, rotated rx 180 ry 0 rz -180 deg; joints [35.732, 33.004, 33.826, -141.956, 71.373, -194.033]
  Call Extruder(33905.894)
  MoveL 3603 to (-49.53, -23.85, 155) mm, rotated rx 180 ry 0 rz 180 deg; joints [33.663, 32.566, 34.615, -144.151, 71.168, -193.128]
  Call Extruder(33916.824)
  MoveL 3604 to (-42.98, -34.27, 155) mm, rotated rx 180 ry 0 rz 180 deg; joints [31.506, 32.553, 34.638, -146.379, 70.7, -192.395]
  Call Extruder(33927.754)
  MoveL 3605 to (-34.27, -42.98, 155) mm, rotated rx 180 ry 0 rz 180 deg; joints [29.427, 32.967, 33.892, -148.473, 69.984, -191.858]
  Call Extruder(33938.684)
  MoveL 3606 to (-23.85, -49.53, 155) mm, rotated rx -180 ry 0 rz 180 deg; joints [27.581, 33.778, 32.428, -150.279, 69.047, -191.538]
  Call Extruder(33949.614)
  MoveL 3607 to (-12.23, -53.59, 155) mm, rotated rx 180 ry 0 rz 180 deg; joints [26.087, 34.935, 30.334, -151.673, 67.929, -191.45]
  Call Extruder(33960.545)
  MoveL 3608 to (0, -54.97, 155) mm, rotated rx 180 ry 0 rz 180 deg; joints [25.019, 36.365, 27.733, -152.579, 66.682, -191.606]
  Call Extruder(33971.475)
  MoveL 3609 to (12.23, -53.59, 155) mm, rotated rx 180 ry 0 rz 180 deg; joints [24.406, 37.99, 24.768, -152.963, 65.364, -192.01]
  Call Extruder(33982.405)
  MoveL 3610 to (23.85, -49.52, 155) mm, rotated rx -180 ry 0 rz -180 deg; joints [24.239, 39.725, 21.589, -152.831, 64.043, -192.661]
  Call Extruder(33993.335)
  MoveL 3611 to (34.27, -42.98, 155) mm, rotated rx 180 ry 0 rz -180 deg; joints [24.487, 41.485, 18.351, -152.22, 62.788, -193.544]
  Call Extruder(34004.265)
  MoveL 3612 to (42.98, -34.27, 155) mm, rotated rx -180 ry 0 rz -180 deg; joints [25.101, 43.19, 15.205, -151.187, 61.668, -194.63]
  Call Extruder(34015.196)
  MoveL 3613 to (49.52, -23.85, 155) mm, rotated rx -180 ry 0 rz 180 deg; joints [26.025, 44.76, 12.299, -149.809, 60.749, -195.87]
  Call Extruder(34026.126)
  MoveL 3614 to (53.59, -12.23, 155) mm, rotated rx 180 ry 0 rz -180 deg; joints [27.2, 46.123, 9.771, -148.172, 60.085, -197.2]
  Call Extruder(34037.056)
  MoveL 3615 to (54.97, 0, 155) mm, rotated rx 180 ry 0 rz -180 deg; joints [28.57, 47.214, 7.745, -146.372, 59.718, -198.54]
  Call Extruder(34047.986)
  MoveL 3616 to (53.59, 12.23, 155) mm, rotated rx 180 ry 0 rz 180 deg; joints [30.077, 47.978, 6.323, -144.506, 59.672, -199.804]
  Call Extruder(34058.916)
  MoveL 3617 to (49.53, 23.85, 155) mm, rotated rx 180 ry 0 rz -180 deg; joints [31.665, 48.377, 5.581, -142.664, 59.948, -200.906]
  Call Extruder(34069.847)
  MoveL 3618 to (42.98, 34.27, 155) mm, rotated rx -180 ry 0 rz -180 deg; joints [33.282, 48.388, 5.56, -140.926, 60.529, -201.774]
  Call Extruder(34080.777)
  MoveL 3619 to (34.27, 42.98, 155) mm, rotated rx 180 ry 0 rz 180 deg; joints [34.874, 48.012, 6.26, -139.354, 61.376, -202.356]
  Call Extruder(34091.707)
  MoveL 3620 to (23.85, 49.53, 155) mm, rotated rx 180 ry 0 rz 180 deg; joints [36.387, 47.269, 7.643, -137.995, 62.435, -202.624]
  Call Extruder(34102.637)
  MoveL 3621 to (12.23, 53.59, 155) mm, rotated rx -180 ry 0 rz -180 deg; joints [37.766, 46.195, 9.637, -136.883, 63.643, -202.573]
  Call Extruder(34113.567)
  MoveL 3622 to (0, 54.97, 155) mm, rotated rx 180 ry 0 rz 180 deg; joints [38.954, 44.846, 12.139, -136.046, 64.931, -202.221]
  Call Extruder(34124.498)
  MoveL 3623 to (-12.23, 53.59, 155) mm, rotated rx -180 ry 0 rz -180 deg; joints [39.895, 43.286, 15.026, -135.508, 66.233, -201.6]
  Call Extruder(34135.428)
  MoveL 3624 to (-23.85, 49.52, 155) mm, rotated rx -180 ry 0 rz -180 deg; joints [40.528, 41.588, 18.161, -135.296, 67.485, -200.756]
  Call Extruder(34146.358)
  MoveL 3625 to (-34.27, 42.98, 155) mm, rotated rx 180 ry 0 rz 180 deg; joints [40.799, 39.828, 21.398, -135.441, 68.63, -199.739]
  Call Extruder(34157.288)
  MoveL 3626 to (-42.98, 34.27, 155) mm, rotated rx -180 ry 0 rz -180 deg; joints [40.659, 38.09, 24.585, -135.968, 69.621, -198.606]
  Call Extruder(34168.218)
  MoveL 3627 to (-49.52, 23.85, 155) mm, rotated rx 180 ry 0 rz -180 deg; joints [40.072, 36.456, 27.567, -136.9, 70.417, -197.414]
  Call Extruder(34179.149)
  MoveL 3628 to (-53.59, 12.23, 155) mm, rotated rx 180 ry 0 rz -180 deg; joints [39.031, 35.012, 30.193, -138.236, 70.988, -196.22]
  Call Extruder(34190.079)
  MoveL 3629 to (-54.97, 0, 155) mm, rotated rx 180 ry 0 rz 180 deg; joints [37.56, 33.837, 32.321, -139.945, 71.311, -195.077]
  Call Extruder(34195.604)
  MoveL 3630 to (-54.27, -6.18, 155) mm, rotated rx 180 ry 0 rz -180 deg; joints [36.644, 33.41, 33.094, -140.954, 71.343, -194.546]
  Set speed (130.0 mm/s)
  MoveL 3631 to (-49.9, -9.51, 155) mm, rotated rx 180 ry 0 rz 180 deg; joints [35.741, 33.62, 32.713, -141.841, 70.985, -194.36]
  MoveL 3632 to (-13.82, -4.91, 155) mm, rotated rx 180 ry 0 rz -180 deg; joints [33.033, 38.067, 24.627, -143.804, 67.382, -195.718]
  Call Extruder(34228.779)
  Set speed (20.0 mm/s)
  MoveL 3633 to (-4.92, -13.82, 155) mm, rotated rx 180 ry 0 rz 180 deg; joints [31.126, 38.462, 23.903, -145.721, 66.606, -195.144]
  Call Extruder(34298.586)
  MoveL 3634 to (13.82, 4.92, 155) mm, rotated rx 180 ry 0 rz -180 deg; joints [32.046, 42.17, 17.087, -143.933, 64.323, -197.515]
  Call Extruder(34331.761)
  MoveL 3635 to (4.92, 13.82, 155) mm, rotated rx 180 ry 0 rz -180 deg; joints [33.834, 41.784, 17.8, -142.143, 65.131, -198.101]
  Set speed (130.0 mm/s)
  MoveL 3636 to (4.92, 13.82, 160) mm, rotated rx 180 ry 0 rz 180 deg; joints [33.834, 41.015, 17.873, -141.942, 64.583, -198.574]
  Call Extruder(34329.761)
  Set speed (40.0 mm/s)
  MoveL 3637 to (4.92, 13.82, 160) mm, rotated rx 180 ry 0 rz 180 deg; joints [33.834, 41.015, 17.873, -141.942, 64.583, -198.574]
  Call Extruder(0.000)
  Set speed (130.0 mm/s)
  MoveL 3638 to (-26.25, -4.54, 160) mm, rotated rx -180 ry 0 rz 180 deg; joints [34.172, 35.81, 27.283, -142.717, 68.012, -195.91]
  Call Extruder(2.000)
  Set speed (40.0 mm/s)
  MoveL 3639 to (-26.25, -4.54, 160) mm, rotated rx -180 ry 0 rz 180 deg; joints [34.172, 35.81, 27.283, -142.717, 68.012, -195.91]
  Call Extruder(4.233)
  Set speed (60.0 mm/s)
  MoveL 3640 to (-26.09, -5.96, 160) mm, rotated rx 180 ry 0 rz 180 deg; joints [33.969, 35.716, 27.45, -142.946, 68.015, -195.783]
  Call Extruder(13.597)
  MoveL 3641 to (-24.11, -11.61, 160) mm, rotated rx 180 ry 0 rz 180 deg; joints [33.033, 35.51, 27.821, -143.959, 67.896, -195.313]
  Call Extruder(22.962)
  MoveL 3642 to (-20.93, -16.69, 160) mm, rotated rx -180 ry 0 rz -180 deg; joints [32.066, 35.504, 27.831, -144.969, 67.647, -194.928]
  Call Extruder(32.328)
  MoveL 3643 to (-16.69, -20.93, 160) mm, rotated rx -180 ry 0 rz -180 deg; joints [31.126, 35.699, 27.482, -145.916, 67.28, -194.646]
  Call Extruder(41.692)
  MoveL 3644 to (-11.61, -24.11, 160) mm, rotated rx -180 ry 0 rz -180 deg; joints [30.272, 36.084, 26.791, -146.742, 66.811, -194.48]
  Call Extruder(51.057)
  MoveL 3645 to (-5.96, -26.09, 160) mm, rotated rx -180 ry 0 rz -180 deg; joints [29.552, 36.637, 25.797, -147.398, 66.261, -194.438]
  Call Extruder(60.422)
  MoveL 3646 to (0, -26.77, 160) mm, rotated rx 180 ry 0 rz -180 deg; joints [29.003, 37.329, 24.552, -147.848, 65.657, -194.526]
  Call Extruder(69.787)
  MoveL 3647 to (5.96, -26.09, 160) mm, rotated rx 180 ry 0 rz -180 deg; joints [28.65, 38.122, 23.121, -148.068, 65.027, -194.742]
  Call Extruder(79.152)
  MoveL 3648 to (11.61, -24.11, 160) mm, rotated rx 180 ry 0 rz -180 deg; joints [28.503, 38.975, 21.577, -148.053, 64.403, -195.078]
  Call Extruder(88.517)
  MoveL 3649 to (16.69, -20.93, 160) mm, rotated rx -180 ry 0 rz -180 deg; joints [28.559, 39.846, 19.998, -147.81, 63.818, -195.523]
  Call Extruder(97.882)
  MoveL 3650 to (20.93, -16.69, 160) mm, rotated rx 180 ry 0 rz -180 deg; joints [28.808, 40.692, 18.46, -147.359, 63.302, -196.055]
  Call Extruder(107.247)
  MoveL 3651 to (24.12, -11.61, 160) mm, rotated rx -180 ry 0 rz -180 deg; joints [29.229, 41.472, 17.041, -146.729, 62.883, -196.651]
  Call Extruder(116.612)
  MoveL 3652 to (26.09, -5.96, 160) mm, rotated rx 180 ry 0 rz 180 deg; joints [29.796, 42.148, 15.809, -145.959, 62.586, -197.278]
  Call Extruder(125.977)
  MoveL 3653 to (26.77, 0, 160) mm, rotated rx 180 ry 0 rz -180 deg; joints [30.482, 42.687, 14.824, -145.092, 62.425, -197.902]
  Call Extruder(135.342)
  MoveL 3654 to (26.09, 5.96, 160) mm, rotated rx 180 ry 0 rz 180 deg; joints [31.252, 43.064, 14.135, -144.171, 62.412, -198.488]
  Call Extruder(144.707)
  MoveL 3655 to (24.11, 11.61, 160) mm, rotated rx 180 ry 0 rz 180 deg; joints [32.076, 43.26, 13.777, -143.242, 62.545, -199.003]
  Call Extruder(154.072)
  MoveL 3656 to (20.93, 16.69, 160) mm, rotated rx 180 ry 0 rz 180 deg; joints [32.917, 43.265, 13.767, -142.346, 62.819, -199.416]
  Call Extruder(163.437)
  MoveL 3657 to (16.69, 20.93, 160) mm, rotated rx 180 ry 0 rz 180 deg; joints [33.742, 43.08, 14.105, -141.522, 63.216, -199.706]
  Call Extruder(172.802)
  MoveL 3658 to (11.61, 24.12, 160) mm, rotated rx 180 ry 0 rz 180 deg; joints [34.517, 42.714, 14.775, -140.802, 63.714, -199.858]
  Call Extruder(182.167)
  MoveL 3659 to (5.96, 26.09, 160) mm, rotated rx 180 ry 0 rz -180 deg; joints [35.208, 42.183, 15.743, -140.214, 64.287, -199.864]
  Call Extruder(191.532)
  MoveL 3660 to (0, 26.77, 160) mm, rotated rx -180 ry 0 rz 180 deg; joints [35.784, 41.515, 16.963, -139.783, 64.904, -199.73]
  Call Extruder(200.897)
  MoveL 3661 to (-5.96, 26.09, 160) mm, rotated rx 180 ry 0 rz 180 deg; joints [36.214, 40.74, 18.373, -139.527, 65.533, -199.463]
  Call Extruder(210.262)
  MoveL 3662 to (-11.61, 24.12, 160) mm, rotated rx 180 ry 0 rz 180 deg; joints [36.473, 39.897, 19.905, -139.459, 66.142, -199.083]
  Call Extruder(219.627)
  MoveL 3663 to (-16.69, 20.93, 160) mm, rotated rx 180 ry 0 rz 180 deg; joints [36.542, 39.026, 21.484, -139.589, 66.703, -198.609]
  Call Extruder(228.992)
  MoveL 3664 to (-20.93, 16.69, 160) mm, rotated rx 180 ry 0 rz 180 deg; joints [36.407, 38.171, 23.033, -139.919, 67.189, -198.068]
  Call Extruder(238.357)
  MoveL 3665 to (-24.12, 11.61, 160) mm, rotated rx 180 ry 0 rz 180 deg; joints [36.065, 37.373, 24.472, -140.442, 67.578, -197.488]
  Call Extruder(247.722)
  MoveL 3666 to (-26.09, 5.96, 160) mm, rotated rx 180 ry 0 rz 180 deg; joints [35.528, 36.674, 25.73, -141.142, 67.853, -196.895]
  Call Extruder(257.087)
  MoveL 3667 to (-26.77, 0, 160) mm, rotated rx 180 ry 0 rz 180 deg; joints [34.817, 36.112, 26.741, -141.99, 68.001, -196.318]
  Call Extruder(261.876)
  MoveL 3668 to (-26.42, -3.05, 160) mm, rotated rx 180 ry 0 rz -180 deg; joints [34.385, 35.908, 27.107, -142.478, 68.008, -196.044]
  Call Extruder(259.876)
  Set speed (40.0 mm/s)
  MoveL 3669 to (-26.42, -3.05, 160) mm, rotated rx 180 ry 0 rz -180 deg; joints [34.385, 35.908, 27.107, -142.478, 68.008, -196.044]
  Call Extruder(0.000)
  Set speed (130.0 mm/s)
  MoveL 3670 to (-41.86, -6.3, 160) mm, rotated rx -180 ry 0 rz -180 deg; joints [35.393, 33.881, 30.73, -141.817, 69.542, -195.37]
  Call Extruder(2.000)
  Set speed (40.0 mm/s)
  MoveL 3671 to (-41.86, -6.3, 160) mm, rotated rx -180 ry 0 rz -180 deg; joints [35.393, 33.881, 30.73, -141.817, 69.542, -195.37]
  Call Extruder(6.998)
  Set speed (60.0 mm/s)
  MoveL 3672 to (-41.5, -9.47, 160) mm, rotated rx -180 ry 0 rz -180 deg; joints [34.924, 33.668, 31.109, -142.338, 69.55, -195.092]
  Call Extruder(21.893)
  MoveL 3673 to (-38.36, -18.47, 160) mm, rotated rx 180 ry 0 rz -180 deg; joints [33.373, 33.331, 31.71, -143.999, 69.366, -194.362]
  Call Extruder(36.789)
  MoveL 3674 to (-33.28, -26.54, 160) mm, rotated rx -180 ry 0 rz -180 deg; joints [31.763, 33.321, 31.727, -145.672, 68.981, -193.763]
  Call Extruder(51.685)
  MoveL 3675 to (-26.54, -33.28, 160) mm, rotated rx 180 ry 0 rz -180 deg; joints [30.206, 33.64, 31.16, -147.243, 68.409, -193.32]
  Call Extruder(66.581)
  MoveL 3676 to (-18.47, -38.36, 160) mm, rotated rx -180 ry 0 rz -180 deg; joints [28.808, 34.267, 30.043, -148.606, 67.675, -193.051]
  Call Extruder(81.477)
  MoveL 3677 to (-9.47, -41.51, 160) mm, rotated rx 180 ry 0 rz 180 deg; joints [27.654, 35.164, 28.439, -149.673, 66.809, -192.972]
  Call Extruder(96.373)
  MoveL 3678 to (0, -42.57, 160) mm, rotated rx 180 ry 0 rz 180 deg; joints [26.805, 36.279, 26.441, -150.383, 65.852, -193.092]
  Call Extruder(111.268)
  MoveL 3679 to (9.47, -41.5, 160) mm, rotated rx 180 ry 0 rz 180 deg; joints [26.29, 37.55, 24.153, -150.705, 64.849, -193.412]
  Call Extruder(126.164)
  MoveL 3680 to (18.47, -38.36, 160) mm, rotated rx 180 ry 0 rz 180 deg; joints [26.114, 38.912, 21.693, -150.636, 63.849, -193.927]
  Call Extruder(141.060)
  MoveL 3681 to (26.54, -33.28, 160) mm, rotated rx -180 ry 0 rz -180 deg; joints [26.262, 40.296, 19.182, -150.197, 62.906, -194.621]
  Call Extruder(155.956)
  MoveL 3682 to (33.28, -26.54, 160) mm, rotated rx -180 ry 0 rz 180 deg; joints [26.703, 41.636, 16.742, -149.429, 62.07, -195.466]
  Call Extruder(170.852)
  MoveL 3683 to (38.36, -18.47, 160) mm, rotated rx -180 ry 0 rz -180 deg; joints [27.4, 42.87, 14.49, -148.385, 61.389, -196.424]
  Call Extruder(185.747)
  MoveL 3684 to (41.51, -9.47, 160) mm, rotated rx 180 ry 0 rz -180 deg; joints [28.309, 43.939, 12.533, -147.132, 60.903, -197.443]
  Call Extruder(200.643)
  MoveL 3685 to (42.57, 0, 160) mm, rotated rx -180 ry 0 rz -180 deg; joints [29.382, 44.793, 10.967, -145.741, 60.641, -198.466]
  Call Extruder(215.539)
  MoveL 3686 to (41.51, 9.47, 160) mm, rotated rx -180 ry 0 rz 180 deg; joints [30.575, 45.39, 9.872, -144.286, 60.619, -199.429]
  Call Extruder(230.435)
  MoveL 3687 to (38.36, 18.47, 160) mm, rotated rx 180 ry 0 rz -180 deg; joints [31.839, 45.701, 9.3, -142.836, 60.839, -200.273]
  Call Extruder(245.331)
  MoveL 3688 to (33.28, 26.54, 160) mm, rotated rx 180 ry 0 rz -180 deg; joints [33.128, 45.71, 9.284, -141.455, 61.287, -200.945]
  Call Extruder(260.226)
  MoveL 3689 to (26.54, 33.29, 160) mm, rotated rx 180 ry 0 rz -180 deg; joints [34.394, 45.416, 9.823, -140.196, 61.935, -201.407]
  Call Extruder(275.122)
  MoveL 3690 to (18.47, 38.36, 160) mm, rotated rx 180 ry 0 rz 180 deg; joints [35.592, 44.835, 10.889, -139.103, 62.745, -201.636]
  Call Extruder(290.018)
  MoveL 3691 to (9.47, 41.5, 160) mm, rotated rx -180 ry 0 rz 180 deg; joints [36.675, 43.996, 12.429, -138.209, 63.669, -201.626]
  Call Extruder(304.914)
  MoveL 3692 to (0, 42.57, 160) mm, rotated rx 180 ry 0 rz 180 deg; joints [37.594, 42.938, 14.365, -137.544, 64.658, -201.386]
  Call Extruder(319.810)
  MoveL 3693 to (-9.47, 41.51, 160) mm, rotated rx 180 ry 0 rz 180 deg; joints [38.304, 41.712, 16.603, -137.132, 65.659, -200.936]
  Call Extruder(334.705)
  MoveL 3694 to (-18.47, 38.36, 160) mm, rotated rx -180 ry 0 rz -180 deg; joints [38.762, 40.376, 19.035, -136.993, 66.622, -200.309]
  Call Extruder(349.601)
  MoveL 3695 to (-26.54, 33.29, 160) mm, rotated rx 180 ry 0 rz 180 deg; joints [38.928, 38.993, 21.545, -137.149, 67.504, -199.542]
  Call Extruder(364.497)
  MoveL 3696 to (-33.28, 26.54, 160) mm, rotated rx 180 ry 0 rz 180 deg; joints [38.772, 37.628, 24.011, -137.611, 68.263, -198.677]
  Call Extruder(379.393)
  MoveL 3697 to (-38.36, 18.47, 160) mm, rotated rx 180 ry 0 rz 180 deg; joints [38.277, 36.35, 26.313, -138.385, 68.869, -197.757]
  Call Extruder(394.288)
  MoveL 3698 to (-41.5, 9.47, 160) mm, rotated rx -180 ry 0 rz -180 deg; joints [37.447, 35.224, 28.332, -139.458, 69.296, -196.826]
  Call Extruder(409.184)
  MoveL 3699 to (-42.57, 0, 160) mm, rotated rx 180 ry 0 rz -180 deg; joints [36.31, 34.313, 29.961, -140.796, 69.526, -195.925]
  Call Extruder(416.739)
  MoveL 3700 to (-42.03, -4.8, 160) mm, rotated rx 180 ry 0 rz 180 deg; joints [35.612, 33.982, 30.55, -141.574, 69.538, -195.501]
  Call Extruder(414.739)
  Set speed (40.0 mm/s)
  MoveL 3701 to (-42.03, -4.8, 160) mm, rotated rx 180 ry 0 rz 180 deg; joints [35.612, 33.982, 30.55, -141.574, 69.538, -195.501]
  Call Extruder(0.000)
  Set speed (130.0 mm/s)
  MoveL 3702 to (-54.1, -7.67, 160) mm, rotated rx 180 ry 0 rz 180 deg; joints [36.421, 32.404, 33.353, -141.021, 70.707, -194.968]
  Call Extruder(2.000)
  Set speed (40.0 mm/s)
  MoveL 3703 to (-54.1, -7.67, 160) mm, rotated rx 180 ry 0 rz 180 deg; joints [36.421, 32.404, 33.353, -141.021, 70.707, -194.968]
  Call Extruder(6.073)
  Set speed (30.0 mm/s)
  MoveL 3704 to (-53.59, -12.23, 160) mm, rotated rx 180 ry 0 rz 180 deg; joints [35.732, 32.093, 33.903, -141.779, 70.718, -194.577]
  Call Extruder(17.003)
  MoveL 3705 to (-49.53, -23.85, 160) mm, rotated rx 180 ry 0 rz -180 deg; joints [33.663, 31.646, 34.693, -143.979, 70.486, -193.651]
  Call Extruder(27.933)
  MoveL 3706 to (-42.98, -34.27, 160) mm, rotated rx 180 ry 0 rz -180 deg; joints [31.506, 31.633, 34.715, -146.212, 69.999, -192.891]
  Call Extruder(38.863)
  MoveL 3707 to (-34.27, -42.98, 160) mm, rotated rx 180 ry 0 rz -180 deg; joints [29.427, 32.055, 33.97, -148.311, 69.273, -192.325]
  Call Extruder(49.793)
  MoveL 3708 to (-23.85, -49.52, 160) mm, rotated rx 180 ry 0 rz -180 deg; joints [27.581, 32.883, 32.505, -150.12, 68.337, -191.975]
  Call Extruder(60.724)
  MoveL 3709 to (-12.23, -53.59, 160) mm, rotated rx 180 ry 0 rz -180 deg; joints [26.087, 34.061, 30.41, -151.516, 67.228, -191.861]
  Call Extruder(71.654)
  MoveL 3710 to (0, -54.97, 160) mm, rotated rx 180 ry 0 rz -180 deg; joints [25.019, 35.517, 27.808, -152.422, 65.996, -191.995]
  Call Extruder(82.584)
  MoveL 3711 to (12.23, -53.59, 160) mm, rotated rx 180 ry 0 rz -180 deg; joints [24.406, 37.168, 24.842, -152.804, 64.698, -192.386]
  Call Extruder(93.514)
  MoveL 3712 to (23.85, -49.52, 160) mm, rotated rx 180 ry 0 rz -180 deg; joints [24.239, 38.928, 21.662, -152.668, 63.4, -193.03]
  Call Extruder(104.444)
  MoveL 3713 to (34.27, -42.98, 160) mm, rotated rx 180 ry 0 rz 180 deg; joints [24.487, 40.713, 18.423, -152.05, 62.17, -193.913]
  Call Extruder(115.375)
  MoveL 3714 to (42.98, -34.27, 160) mm, rotated rx 180 ry 0 rz -180 deg; joints [25.101, 42.439, 15.277, -151.008, 61.074, -195.003]
  Call Extruder(126.305)
  MoveL 3715 to (49.52, -23.85, 160) mm, rotated rx 180 ry 0 rz -180 deg; joints [26.025, 44.027, 12.372, -149.62, 60.179, -196.253]
  Call Extruder(137.235)
  MoveL 3716 to (53.59, -12.23, 160) mm, rotated rx 180 ry 0 rz -180 deg; joints [27.2, 45.405, 9.844, -147.974, 59.537, -197.595]
  Call Extruder(148.165)
  MoveL 3717 to (54.97, 0, 160) mm, rotated rx 180 ry 0 rz 180 deg; joints [28.57, 46.507, 7.818, -146.164, 59.191, -198.949]
  Call Extruder(159.095)
  MoveL 3718 to (53.59, 12.23, 160) mm, rotated rx -180 ry 0 rz 180 deg; joints [30.077, 47.278, 6.396, -144.29, 59.162, -200.228]
  Call Extruder(170.026)
  MoveL 3719 to (49.53, 23.85, 160) mm, rotated rx 180 ry 0 rz 180 deg; joints [31.665, 47.681, 5.654, -142.443, 59.453, -201.345]
  Call Extruder(180.956)
  MoveL 3720 to (42.98, 34.27, 160) mm, rotated rx 180 ry 0 rz 180 deg; joints [33.282, 47.692, 5.633, -140.701, 60.046, -202.228]
  Call Extruder(191.886)
  MoveL 3721 to (34.27, 42.98, 160) mm, rotated rx 180 ry 0 rz 180 deg; joints [34.874, 47.313, 6.333, -139.128, 60.901, -202.824]
  Call Extruder(202.816)
  MoveL 3722 to (23.85, 49.53, 160) mm, rotated rx -180 ry 0 rz -180 deg; joints [36.387, 46.562, 7.716, -137.77, 61.964, -203.105]
  Call Extruder(213.746)
  MoveL 3723 to (12.23, 53.59, 160) mm, rotated rx 180 ry 0 rz 180 deg; joints [37.766, 45.478, 9.709, -136.662, 63.173, -203.067]
  Call Extruder(224.677)
  MoveL 3724 to (0, 54.97, 160) mm, rotated rx 180 ry 0 rz -180 deg; joints [38.954, 44.115, 12.211, -135.829, 64.457, -202.728]
  Call Extruder(235.607)
  MoveL 3725 to (-12.23, 53.59, 160) mm, rotated rx 180 ry 0 rz -180 deg; joints [39.895, 42.537, 15.099, -135.296, 65.751, -202.121]
  Call Extruder(246.537)
  MoveL 3726 to (-23.85, 49.53, 160) mm, rotated rx 180 ry 0 rz -180 deg; joints [40.528, 40.817, 18.234, -135.09, 66.99, -201.289]
  Call Extruder(257.467)
  MoveL 3727 to (-34.27, 42.98, 160) mm, rotated rx 180 ry 0 rz 180 deg; joints [40.799, 39.034, 21.472, -135.24, 68.117, -200.285]
  Call Extruder(268.397)
  MoveL 3728 to (-42.98, 34.27, 160) mm, rotated rx 180 ry 0 rz -180 deg; joints [40.659, 37.269, 24.659, -135.773, 69.085, -199.161]
  Call Extruder(279.328)
  MoveL 3729 to (-49.53, 23.85, 160) mm, rotated rx 180 ry 0 rz 180 deg; joints [40.072, 35.609, 27.642, -136.709, 69.854, -197.976]
  Call Extruder(290.258)
  MoveL 3730 to (-53.59, 12.23, 160) mm, rotated rx 180 ry 0 rz -180 deg; joints [39.031, 34.14, 30.269, -138.049, 70.395, -196.783]
  Call Extruder(301.188)
  MoveL 3731 to (-54.97, 0, 160) mm, rotated rx -180 ry 0 rz 180 deg; joints [37.56, 32.943, 32.398, -139.763, 70.686, -195.635]
  Call Extruder(306.714)
  MoveL 3732 to (-54.27, -6.18, 160) mm, rotated rx 180 ry 0 rz 180 deg; joints [36.644, 32.507, 33.171, -140.774, 70.703, -195.097]
  Set speed (130.0 mm/s)
  MoveL 3733 to (-49.9, -9.51, 160) mm, rotated rx 180 ry 0 rz 180 deg; joints [35.741, 32.722, 32.79, -141.663, 70.34, -194.899]
  Call Extruder(304.714)
  Set speed (40.0 mm/s)
  MoveL 3734 to (-49.9, -9.51, 160) mm, rotated rx 180 ry 0 rz 180 deg; joints [35.741, 32.722, 32.79, -141.663, 70.34, -194.899]
  Call Extruder(0.000)
  Set speed (130.0 mm/s)
  MoveL 3735 to (-4.91, 13.82, 160) mm, rotated rx 180 ry 0 rz -180 deg; joints [34.648, 39.818, 20.049, -141.372, 65.608, -198.263]
  Call Extruder(2.000)
  Set speed (40.0 mm/s)
  MoveL 3736 to (-4.91, 13.82, 160) mm, rotated rx 180 ry 0 rz -180 deg; joints [34.648, 39.818, 20.049, -141.372, 65.608, -198.263]
  Call Extruder(35.175)
  Set speed (15.0 mm/s)
  MoveL 3737 to (-13.82, 4.91, 160) mm, rotated rx 180 ry 0 rz 180 deg; joints [34.301, 38.025, 23.296, -142.133, 66.644, -197.133]
  Call Extruder(104.982)
  MoveL 3738 to (4.91, -13.82, 160) mm, rotated rx 180 ry 0 rz 180 deg; joints [30.357, 38.863, 21.78, -146.1, 64.974, -195.869]
  Call Extruder(138.157)
  MoveL 3739 to (13.82, -4.91, 160) mm, rotated rx 180 ry 0 rz 180 deg; joints [30.824, 40.646, 18.545, -145.212, 63.907, -196.991]
  Call Extruder(136.157)
  Set speed (40.0 mm/s)
  MoveL 3740 to (13.82, -4.91, 160) mm, rotated rx 180 ry 0 rz 180 deg; joints [30.824, 40.646, 18.545, -145.212, 63.907, -196.991]
  Set speed (1000.0 mm/s)
  Call Extruder(-1)
  MoveL 3741 to (13.82, -4.91, 160) mm, rotated rx 180 ry 0 rz 180 deg; joints [30.824, 40.646, 18.545, -145.212, 63.907, -196.991]
  Call Extruder(0.000)

--- Python program Extruder ---
# This macro allows simulating a 3D printing extruder
# The macro will output spray gun statistics
#
# More information about the RoboDK API here:
# https://robodk.com/doc/en/RoboDK-API.html
# For more information visit:
# http://www.robodk.com/doc/en/PythonAPI/robolink.html
#
# Define the default action (0 to deactivate, +1 to activate, -1 to clear any spray gun simulation)
# Setting it to None will display a message
ACTION = None
# Check if we are running this program inside another program and passing arguments
import sys
if len(sys.argv) > 1:
    ACTION = float(sys.argv[1])
    # For faster speed: igone values greater than 0
    if ACTION > 0:
        quit()

from robolink import *    # API to communicate with RoboDK
from robodk import *      # basic matrix operations
RDK = Robolink()

# quit if we are not in simulation mode
if RDK.RunMode() != RUNMODE_SIMULATE:
    quit()

# Get any previously added spray gun simulations and display statistics (spray on the part vs spray falling out of the part)
existing_material_simulation = False
info, stats_data = RDK.Spray_GetStats()
if stats_data.size(1) > 0:
    print("Spray gun statistics:")
    print(info)
    print(stats_data.tr())
    existing_material_simulation = True
    # # Diplay statistics
    # RDK.ShowMessage("Material used: %.1f%%<br>Material waisted: %.1f%%<br>Total particles: %.1f" % (data[1,0],data[2,0],data[3,0]), True)
    # # Clear previous spray
    # RDK.Spray_Clear()

# If the default ACTION is None, display a message to activate/deactivate the spray gun
if ACTION is None:
    print('Note: This macro can be called as Extruder(0) to turn it ON or Extruder(-1) to turn it OFF')
    entry = mbox('Turn Extruder ON or OFF', ('On', '0'), ('Off', '-1'))
    if not entry:
        quit()
    ACTION = int(entry)

if ACTION < 0:
    # Turn material deposition off
    # Select Escape to delete existing material simulations
    #RDK.Spray_Clear()
    RDK.Spray_SetState(SPRAY_OFF)

elif ACTION >= 0:

    if existing_material_simulation:
        # Select Esc key to delete existing material simulations and force a new type of spray gun simulation
        RDK.Spray_SetState(SPRAY_ON)
        exit()


    # Create a new spray gun object in RoboDK for material deposition (3D printing simulation)
    # by using RDK.Spray_Add(tool, object, options_command, volume, geometry)
    # tool: tool item (TCP) to use
    # object: object to project the particles
    # options_command (optional): string to specify options. Example:
    #     STEP=AxB: Defines the grid to be projected 1x1 means only one line of particle projection (for example, for welding)
    #     PARTICLE: Defines the shape and size of particle (sphere or particle), unless a specific geometry is provided:
    #       a- SPHERE(radius, facets)
    #       b- SPHERE(radius, facets, scalex, scaley, scalez)
    #       b- CUBE(sizex, sizey, sizez)
    #     RAND=factor: Defines a random factor factor 0 means that the particles are not deposited randomly
    #     ELLYPSE: defines the volume as an ellypse (default)
    #     RECTANGLE: defines the volume as a rectangle
    #     PROJECT: project the particles to the surface (default) (for welding, painting or scanning)
    #     NO_PROJECT: does not project the particles to the surface (for example, for 3D printing)
    #
    # volume (optional): Matrix of parameters defining the volume of the spray gun
    # geometry (optional): Matrix of vertices defining the triangles.


    diameter = 10 # in mm
    detail = 8 # number of rings of detail to display the sphere
    scale = '1,1,0.5' # scale the particle in 0.5 along the tool Z axis (simulating gravity effect)
    options_command = "ELLYPSE NO_PROJECT PARTICLE=SPHERE(%.3f,%.0f,%s)" % (diameter, detail, scale) # simulate
    #options_command = "PARTICLE=CUBE(10,10,2) STEP=8x8"
    #options_command = "PARTICLE=SPHERE(4,8) STEP=8x8"
    #options_command = "PARTICLE=SPHERE(4,8,1,1,0.1) STEP=8x8 RAND=3"

    # Example commands for welding:
    # options_command = "PROJECT PARTICLE=SPHERE(4,8)"
    # options_command = PARTICLE=SPHERE(4,8) STEP=1x0

    tool = 0    # auto detect active tool
    obj = 0     # auto detect object in active reference frame

    # Material is deposited at 0,0,0 with respect to the TCP coordinates
    close_param = [0,0,0,  0,0,0,  0,0,0,     0.7,0.5,0.8,1] # color as RGBA
    far_param   = [0,0,0,  0,0,0,  0,0,0,     0.7,0.5,0.8,1] # color as RGBA
    volume = Mat([close_param, far_param])
    RDK.Spray_Add(tool, obj, options_command, volume.tr())
    RDK.Spray_SetState(SPRAY_ON)

--- Python program SimulateFinalResult ---
# This script will simulate the final result of the 3D printed part using the Spray function

# Or visit: http://www.robodk.com/doc/PythonAPI/
# Note: you do not need to keep a copy of this file, your python script is saved with the station
from robolink import *    # API to communicate with RoboDK
from robodk import *      # basic matrix operations


RENDER = True      # Set to False
STEP_MM = 2         # Detail step in MM for linear moves
STEP_DEG = 2        # Detail step in DEG for joint moves

# Start a connection with the RoboDK API
RDK = Robolink()

# Select the first/only robot in the cell:
program = RDK.ItemUserPick('Select a program to simulate', ITEM_TYPE_PROGRAM)
if not program.Valid():
    raise Exception("No program available")

# Get the robot
robot = RDK.Item('', ITEM_TYPE_ROBOT)
#robot = program.getLink(ITEM_TYPE_ROBOT) # available in newer versions
if not robot.Valid():
    raise Exception("No robot available")

progname = program.Name()
print("Using program %s" % progname)


# Get the program as a list of joint values
tool = robot.getLink(ITEM_TYPE_TOOL)
progok_jlist = program.InstructionListJoints(STEP_MM, STEP_DEG)
progok = progok_jlist[0] # progok: String that indicates if there are any issues with the program
jlist = progok_jlist[1]  # jlist: list of joints

# Check that the program is correct and has at least a movement
njoints = jlist.size(1)
if njoints < 1:
    raise Exception("Program %s has no movements" % name)

# Check if there are any issues with the program:
if progok != "Success":
    raise Exception("Problems with program %s: %s." %(name, progok))

# Reset any material deposition simulation
RDK.Spray_Clear()

robot.setPoseTool(tool)

# Start material deposition simulation according to the Extruder script
RDK.RunProgram('Extruder(0)')
# Alternatively:
#RDK.Item('Extruder', ITEM_TYPE_PYTHON).RunProgram([1])

